KUKA KRL program: Machining.src

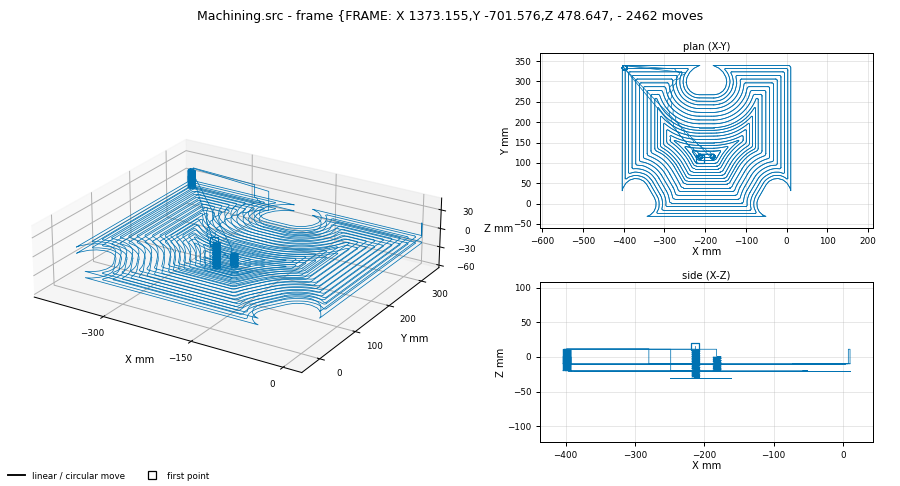
[picture p0: tool path of Machining.src in frame {FRAME: X 1373.155,Y -701.576,Z 478.647,, 2462 of 2464 moves have a stored position in this frame; points joined in program order, loops and branches not executed]
&ACCESS RVP
&REL 1
&PARAM TEMPLATE = C:\KRC\Roboter\Template\vorgabe
&PARAM EDITMASK = *
DEF Machining ( )

; External program calls:
EXT Machining1()


EXT BAS (BAS_COMMAND :IN,REAL :IN )

;FOLD INI
BAS (#INITMOV,0 )
;ENDFOLD (INI)

;FOLD STARTPOS
$BWDSTART = FALSE
PDAT_ACT = PDEFAULT
BAS(#PTP_DAT)
FDAT_ACT = {TOOL_NO 0,BASE_NO 0,IPO_FRAME #BASE}
BAS(#FRAMES)
;ENDFOLD

;FOLD SET DEFAULT SPEED
$VEL.CP=0.2
BAS(#VEL_PTP,100)
BAS(#TOOL,0)
BAS(#BASE,0)
;ENDFOLD

$ADVANCE = 5

PTP $AXIS_ACT ; skip BCO quickly

; Program generated by RoboDK v3.5.4 for GIGASHEEN on 08/07/2019 07:57:20
; Using nominal kinematics.
$APO.CPTP = 1.000
$APO.CDIS = 1.000
$BASE = {FRAME: X 1373.155,Y -701.576,Z 478.647,A -180.000,B 0.620,C 1.380}
$TOOL = {FRAME: X 337.715,Y -2.199,Z 160.575,A 0.000,B 90.000,C 0.000}
; Show 1/2" End Mill TCP
Wait for StrClear($LOOP_MSG[])
$LOOP_CONT = TRUE
$LOOP_MSG[] = "/'1001'"
Wait for StrClear($LOOP_MSG[])
$LOOP_CONT = TRUE
$LOOP_MSG[] = "/''"
Wait for StrClear($LOOP_MSG[])
$LOOP_CONT = TRUE
$LOOP_MSG[] = "/'Pocket2'"
$VEL.CP = 1.00000
$VEL.CP = 1.00000
PTP {A1 32.59641,A2 -47.79719,A3 105.13818,A4 -142.99270,A5 63.54911,A6 162.42451} C_PTP
LIN {X -212.831,Y 109.367,Z 15.000,A 0.015,B 0.000,C 180.000} C_DIS
LIN {X -212.831,Y 109.367,Z 15.000,A 0.015,B 0.000,C 180.000} C_DIS
$VEL.CP = 1.00000
LIN {X -212.831,Y 109.367,Z 11.769,A 0.015,B 0.000,C 180.000} C_DIS
$VEL.CP = 0.10000
LIN {X -212.669,Y 109.348,Z 11.147,A 0.015,B 0.000,C -180.000} C_DIS
LIN {X -212.223,Y 109.320,Z 10.684,A 0.015,B 0.000,C -180.000} C_DIS
LIN {X -211.608,Y 109.335,Z 10.500,A 0.015,B -0.000,C 180.000} C_DIS
LIN {X -206.370,Y 113.359,Z 10.256,A 0.015,B 0.000,C -180.000} C_DIS
LIN {X -207.958,Y 119.769,Z 10.012,A 0.015,B 0.000,C -180.000} C_DIS
LIN {X -214.467,Y 120.884,Z 9.768,A 0.015,B 0.000,C -180.000} C_DIS
LIN {X -218.097,Y 115.366,Z 9.524,A 0.015,B 0.000,C -180.000} C_DIS
LIN {X -214.496,Y 109.830,Z 9.280,A 0.015,B 0.000,C 180.000} C_DIS
LIN {X -207.981,Y 110.910,Z 9.036,A 0.015,B 0.000,C 180.000} C_DIS
LIN {X -206.360,Y 117.312,Z 8.792,A 0.015,B -0.000,C 180.000} C_DIS
LIN {X -211.576,Y 121.363,Z 8.548,A 0.015,B 0.000,C 180.000} C_DIS
LIN {X -217.378,Y 118.207,Z 8.304,A 0.015,B 0.000,C -180.000} C_DIS
LIN {X -216.811,Y 111.627,Z 8.060,A 0.015,B 0.000,C 180.000} C_DIS
LIN {X -210.555,Y 109.510,Z 7.815,A 0.015,B 0.000,C 180.000} C_DIS
LIN {X -206.108,Y 114.393,Z 7.571,A 0.015,B 0.000,C -180.000} C_DIS
LIN {X -208.800,Y 120.423,Z 7.327,A 0.015,B 0.000,C 180.000} C_DIS
LIN {X -215.404,Y 120.374,Z 7.083,A 0.015,B 0.000,C 180.000} C_DIS
LIN {X -218.005,Y 114.303,Z 6.839,A 0.015,B 0.000,C 180.000} C_DIS
LIN {X -213.486,Y 109.488,Z 6.595,A 0.015,B 0.000,C -180.000} C_DIS
LIN {X -207.263,Y 111.699,Z 6.351,A 0.015,B 0.000,C 180.000} C_DIS
LIN {X -206.795,Y 118.286,Z 6.107,A 0.015,B 0.000,C 180.000} C_DIS
LIN {X -212.643,Y 121.355,Z 5.863,A 0.015,B 0.000,C -180.000} C_DIS
LIN {X -217.798,Y 117.227,Z 5.619,A 0.015,B 0.000,C 180.000} C_DIS
LIN {X -216.081,Y 110.849,Z 5.375,A 0.015,B 0.000,C -180.000} C_DIS
LIN {X -209.550,Y 109.867,Z 5.131,A 0.015,B 0.000,C -180.000} C_DIS
LIN {X -206.033,Y 115.457,Z 4.887,A 0.015,B 0.000,C 180.000} C_DIS
LIN {X -209.745,Y 120.919,Z 4.643,A 0.015,B -0.000,C 180.000} C_DIS
LIN {X -216.237,Y 119.707,Z 4.399,A 0.015,B 0.000,C -180.000} C_DIS
LIN {X -217.728,Y 113.273,Z 4.155,A 0.015,B 0.000,C -180.000} C_DIS
LIN {X -212.431,Y 109.329,Z 3.911,A 0.015,B 0.000,C 180.000} C_DIS
LIN {X -206.695,Y 112.602,Z 3.667,A 0.015,B 0.000,C 180.000} C_DIS
LIN {X -207.394,Y 119.169,Z 3.423,A 0.015,B 0.000,C 180.000} C_DIS
LIN {X -213.691,Y 121.159,Z 3.179,A 0.015,B -0.000,C 180.000} C_DIS
LIN {X -218.039,Y 116.188,Z 2.935,A 0.015,B 0.000,C 180.000} C_DIS
LIN {X -215.225,Y 110.212,Z 2.690,A 0.015,B -0.000,C -180.000} C_DIS
LIN {X -208.624,Y 110.395,Z 2.446,A 0.015,B -0.000,C -180.000} C_DIS
LIN {X -206.146,Y 116.517,Z 2.202,A 0.015,B 0.000,C -180.000} C_DIS
LIN {X -210.762,Y 121.241,Z 1.958,A 0.015,B 0.000,C -180.000} C_DIS
LIN {X -216.939,Y 118.904,Z 1.714,A 0.015,B -0.000,C -180.000} C_DIS
LIN {X -217.274,Y 112.308,Z 1.470,A 0.015,B 0.000,C 180.000} C_DIS
LIN {X -211.365,Y 109.359,Z 1.226,A 0.015,B 0.000,C -180.000} C_DIS
LIN {X -206.294,Y 113.590,Z 0.982,A 0.015,B 0.000,C 180.000} C_DIS
LIN {X -208.140,Y 119.932,Z 0.738,A 0.015,B -0.000,C 180.000} C_DIS
LIN {X -214.689,Y 120.782,Z 0.494,A 0.015,B 0.000,C -180.000} C_DIS
LIN {X -218.093,Y 115.122,Z 0.250,A 0.015,B 0.000,C -180.000} C_DIS
LIN {X -214.271,Y 109.736,Z 0.006,A 0.015,B 0.000,C 180.000} C_DIS
LIN {X -207.805,Y 111.079,Z -0.238,A 0.015,B 0.000,C 180.000} C_DIS
LIN {X -206.444,Y 117.541,Z -0.482,A 0.015,B -0.000,C 180.000} C_DIS
LIN {X -211.820,Y 121.378,Z -0.726,A 0.015,B -0.000,C 180.000} C_DIS
LIN {X -217.489,Y 117.990,Z -0.970,A 0.015,B 0.000,C -180.000} C_DIS
LIN {X -216.657,Y 111.438,Z -1.214,A 0.015,B 0.000,C -180.000} C_DIS
LIN {X -210.320,Y 109.575,Z -1.458,A 0.015,B 0.000,C -180.000} C_DIS
LIN {X -206.075,Y 114.634,Z -1.702,A 0.015,B 0.000,C 180.000} C_DIS
LIN {X -209.008,Y 120.551,Z -1.946,A 0.015,B -0.000,C 180.000} C_DIS
LIN {X -215.605,Y 120.235,Z -2.190,A 0.015,B -0.000,C -180.000} C_DIS
LIN {X -217.958,Y 114.064,Z -2.435,A 0.015,B 0.000,C 180.000} C_DIS
LIN {X -213.248,Y 109.435,Z -2.679,A 0.015,B 0.000,C -180.000} C_DIS
LIN {X -207.119,Y 111.896,Z -2.923,A 0.015,B 0.000,C -180.000} C_DIS
LIN {X -206.918,Y 118.497,Z -3.167,A 0.015,B 0.000,C -180.000} C_DIS
LIN {X -212.885,Y 121.327,Z -3.411,A 0.015,B 0.000,C 180.000} C_DIS
LIN {X -217.869,Y 116.993,Z -3.655,A 0.015,B 0.000,C -180.000} C_DIS
LIN {X -215.896,Y 110.691,Z -3.899,A 0.015,B 0.000,C -180.000} C_DIS
LIN {X -209.331,Y 109.973,Z -4.143,A 0.015,B -0.000,C -180.000} C_DIS
LIN {X -206.042,Y 115.700,Z -4.387,A 0.015,B -0.000,C -180.000} C_DIS
LIN {X -209.972,Y 121.008,Z -4.631,A 0.015,B 0.000,C 180.000} C_DIS
LIN {X -216.410,Y 119.535,Z -4.875,A 0.015,B 0.000,C -180.000} C_DIS
LIN {X -217.640,Y 113.046,Z -5.119,A 0.015,B 0.000,C -180.000} C_DIS
LIN {X -212.187,Y 109.319,Z -5.363,A 0.015,B 0.000,C -180.000} C_DIS
LIN {X -206.588,Y 112.821,Z -5.607,A 0.015,B 0.000,C 180.000} C_DIS
LIN {X -207.552,Y 119.354,Z -5.851,A 0.015,B 0.000,C -180.000} C_DIS
LIN {X -213.925,Y 121.089,Z -6.095,A 0.015,B 0.000,C -180.000} C_DIS
LIN {X -218.068,Y 115.945,Z -6.339,A 0.015,B 0.000,C -180.000} C_DIS
LIN {X -215.015,Y 110.089,Z -6.583,A 0.015,B -0.000,C 180.000} C_DIS
LIN {X -208.426,Y 110.539,Z -6.827,A 0.015,B 0.000,C -180.000} C_DIS
LIN {X -206.198,Y 116.756,Z -7.071,A 0.015,B 0.000,C 180.000} C_DIS
LIN {X -211.001,Y 121.288,Z -7.315,A 0.015,B 0.000,C 180.000} C_DIS
LIN {X -217.079,Y 118.704,Z -7.560,A 0.015,B -0.000,C -180.000} C_DIS
LIN {X -217.147,Y 112.100,Z -7.804,A 0.015,B -0.000,C -180.000} C_DIS
LIN {X -211.123,Y 109.392,Z -8.048,A 0.015,B 0.000,C -180.000} C_DIS
LIN {X -206.228,Y 113.825,Z -8.292,A 0.015,B 0.000,C -180.000} C_DIS
LIN {X -208.328,Y 120.087,Z -8.536,A 0.015,B -0.000,C -180.000} C_DIS
LIN {X -214.907,Y 120.671,Z -8.780,A 0.015,B 0.000,C -180.000} C_DIS
LIN {X -218.078,Y 114.879,Z -9.024,A 0.015,B -0.000,C -180.000} C_DIS
LIN {X -214.042,Y 109.651,Z -9.268,A 0.015,B 0.000,C 180.000} C_DIS
LIN {X -207.636,Y 111.255,Z -9.512,A 0.015,B 0.000,C 180.000} C_DIS
LIN {X -206.537,Y 117.767,Z -9.756,A 0.015,B 0.000,C -180.000} C_DIS
LIN {X -212.064,Y 121.383,Z -10.000,A 0.015,B 0.000,C -180.000} C_DIS
LIN {X -213.992,Y 121.383,Z -10.000,A 0.015,B 0.000,C -180.000} C_DIS
CIRC {X -215.914,Y 120.274,Z -10.000,A 0.015,B 0.000,C 180.000},{X -215.915,Y 118.055,Z -10.000,A 0.015,B 0.000,C -180.000} C_DIS
LIN {X -214.810,Y 116.136,Z -10.000,A 0.015,B -0.000,C -180.000} C_DIS
CIRC {X -213.771,Y 115.096,Z -10.000,A 0.015,B 0.000,C 180.000},{X -212.350,Y 114.715,Z -10.000,A 0.015,B 0.000,C 180.000} C_DIS
LIN {X -181.148,Y 114.715,Z -10.000,A 0.015,B 0.000,C 180.000} C_DIS
CIRC {X -179.729,Y 115.095,Z -10.000,A 0.015,B -0.000,C 180.000},{X -178.690,Y 116.133,Z -10.000,A 0.015,B 0.000,C -180.000} C_DIS
LIN {X -177.582,Y 118.050,Z -10.000,A 0.015,B 0.000,C 180.000} C_DIS
CIRC {X -177.581,Y 120.268,Z -10.000,A 0.015,B 0.000,C -180.000},{X -179.502,Y 121.378,Z -10.000,A 0.015,B 0.000,C -180.000} C_DIS
LIN {X -212.064,Y 121.383,Z -10.000,A 0.015,B 0.000,C -180.000} C_DIS
CIRC {X -215.545,Y 122.470,Z -10.000,A 0.015,B 0.000,C 180.000},{X -217.792,Y 125.344,Z -10.000,A 0.015,B -0.000,C -180.000} C_DIS
CIRC {X -219.970,Y 128.243,Z -10.000,A 0.015,B 0.000,C 180.000},{X -223.364,Y 129.521,Z -10.000,A 0.015,B 0.000,C 180.000} C_DIS
CIRC {X -226.438,Y 129.779,Z -10.000,A 0.015,B 0.000,C -180.000},{X -229.509,Y 130.077,Z -10.000,A 0.015,B 0.000,C -180.000} C_DIS
CIRC {X -231.315,Y 129.159,Z -10.000,A 0.015,B 0.000,C -180.000},{X -231.219,Y 127.135,Z -10.000,A 0.015,B 0.000,C 180.000} C_DIS
CIRC {X -228.507,Y 123.213,Z -10.000,A 0.015,B 0.000,C 180.000},{X -225.924,Y 119.206,Z -10.000,A 0.015,B -0.000,C 180.000} C_DIS
CIRC {X -223.440,Y 115.136,Z -10.000,A 0.015,B 0.000,C 180.000},{X -221.024,Y 111.025,Z -10.000,A 0.015,B 0.000,C -180.000} C_DIS
CIRC {X -217.920,Y 107.917,Z -10.000,A 0.015,B -0.000,C 180.000},{X -213.676,Y 106.779,Z -10.000,A 0.015,B 0.000,C 180.000} C_DIS
LIN {X -179.836,Y 106.779,Z -10.000,A 0.015,B 0.000,C 180.000} C_DIS
CIRC {X -175.587,Y 107.917,Z -10.000,A 0.015,B 0.000,C 180.000},{X -172.475,Y 111.026,Z -10.000,A 0.015,B 0.000,C -180.000} C_DIS
CIRC {X -170.064,Y 115.135,Z -10.000,A 0.015,B 0.000,C 180.000},{X -167.600,Y 119.211,Z -10.000,A 0.015,B 0.000,C 180.000} C_DIS
CIRC {X -165.032,Y 123.224,Z -10.000,A 0.015,B 0.000,C 180.000},{X -162.314,Y 127.136,Z -10.000,A 0.015,B 0.000,C 180.000} C_DIS
CIRC {X -162.208,Y 129.160,Z -10.000,A 0.015,B 0.000,C 180.000},{X -164.009,Y 130.087,Z -10.000,A 0.015,B 0.000,C -180.000} C_DIS
CIRC {X -167.842,Y 129.694,Z -10.000,A 0.015,B 0.000,C -180.000},{X -171.671,Y 129.271,Z -10.000,A 0.015,B 0.000,C 180.000} C_DIS
CIRC {X -175.512,Y 128.943,Z -10.000,A 0.015,B -0.000,C -180.000},{X -179.364,Y 128.834,Z -10.000,A 0.015,B 0.000,C 180.000} C_DIS
LIN {X -205.629,Y 128.838,Z -10.000,A 0.015,B 0.000,C -180.000} C_DIS
CIRC {X -214.503,Y 129.009,Z -10.000,A 0.015,B 0.000,C -180.000},{X -223.364,Y 129.521,Z -10.000,A 0.015,B 0.000,C -180.000} C_DIS
CIRC {X -226.590,Y 130.783,Z -10.000,A 0.015,B 0.000,C 180.000},{X -228.564,Y 133.630,Z -10.000,A 0.015,B -0.000,C -180.000} C_DIS
CIRC {X -230.489,Y 136.492,Z -10.000,A 0.015,B 0.000,C -180.000},{X -233.646,Y 137.883,Z -10.000,A 0.015,B 0.000,C -180.000} C_DIS
CIRC {X -239.011,Y 138.684,Z -10.000,A 0.015,B -0.000,C -180.000},{X -244.350,Y 139.648,Z -10.000,A 0.015,B 0.000,C 180.000} C_DIS
CIRC {X -245.188,Y 139.826,Z -10.000,A 0.015,B 0.000,C 180.000},{X -246.019,Y 140.030,Z -10.000,A 0.015,B 0.000,C 180.000} C_DIS
CIRC {X -246.851,Y 140.234,Z -10.000,A 0.015,B 0.000,C -180.000},{X -247.688,Y 140.411,Z -10.000,A 0.015,B -0.000,C 180.000} C_DIS
CIRC {X -249.425,Y 139.627,Z -10.000,A 0.015,B 0.000,C -180.000},{X -249.254,Y 137.730,Z -10.000,A 0.015,B 0.000,C -180.000} C_DIS
CIRC {X -245.418,Y 133.290,Z -10.000,A 0.015,B 0.000,C 180.000},{X -241.535,Y 128.891,Z -10.000,A 0.015,B -0.000,C 180.000} C_DIS
CIRC {X -237.771,Y 124.386,Z -10.000,A 0.015,B 0.000,C -180.000},{X -234.304,Y 119.648,Z -10.000,A 0.015,B -0.000,C 180.000} C_DIS
CIRC {X -231.839,Y 115.776,Z -10.000,A 0.015,B 0.000,C -180.000},{X -229.634,Y 111.750,Z -10.000,A 0.015,B 0.000,C 180.000} C_DIS
CIRC {X -227.507,Y 107.684,Z -10.000,A 0.015,B 0.000,C -180.000},{X -225.271,Y 103.678,Z -10.000,A 0.015,B 0.000,C 180.000} C_DIS
CIRC {X -222.166,Y 100.569,Z -10.000,A 0.015,B 0.000,C 180.000},{X -217.922,Y 99.431,Z -10.000,A 0.015,B -0.000,C 180.000} C_DIS
LIN {X -175.596,Y 99.431,Z -10.000,A 0.015,B 0.000,C -180.000} C_DIS
CIRC {X -171.347,Y 100.569,Z -10.000,A 0.015,B -0.000,C 180.000},{X -168.235,Y 103.679,Z -10.000,A 0.015,B 0.000,C -180.000} C_DIS
CIRC {X -164.238,Y 110.524,Z -10.000,A 0.015,B 0.000,C -180.000},{X -160.181,Y 117.333,Z -10.000,A 0.015,B 0.000,C 180.000} C_DIS
CIRC {X -155.834,Y 123.968,Z -10.000,A 0.015,B 0.000,C 180.000},{X -150.994,Y 130.253,Z -10.000,A 0.015,B 0.000,C -180.000} C_DIS
CIRC {X -149.353,Y 132.160,Z -10.000,A 0.015,B -0.000,C 180.000},{X -147.652,Y 134.012,Z -10.000,A 0.015,B 0.000,C -180.000} C_DIS
CIRC {X -145.937,Y 135.852,Z -10.000,A 0.015,B 0.000,C 180.000},{X -144.257,Y 137.724,Z -10.000,A 0.015,B 0.000,C -180.000} C_DIS
CIRC {X -144.062,Y 139.614,Z -10.000,A 0.015,B 0.000,C 180.000},{X -145.784,Y 140.416,Z -10.000,A 0.015,B 0.000,C 180.000} C_DIS
CIRC {X -154.123,Y 138.916,Z -10.000,A 0.015,B 0.000,C 180.000},{X -162.475,Y 137.498,Z -10.000,A 0.015,B -0.000,C -180.000} C_DIS
CIRC {X -170.891,Y 136.464,Z -10.000,A 0.015,B 0.000,C -180.000},{X -179.363,Y 136.119,Z -10.000,A 0.015,B 0.000,C -180.000} C_DIS
LIN {X -211.942,Y 136.310,Z -10.000,A 0.015,B 0.000,C -180.000} C_DIS
CIRC {X -222.818,Y 136.767,Z -10.000,A 0.015,B 0.000,C -180.000},{X -233.646,Y 137.883,Z -10.000,A 0.015,B 0.000,C -180.000} C_DIS
CIRC {X -236.389,Y 139.137,Z -10.000,A 0.015,B 0.000,C -180.000},{X -237.966,Y 141.708,Z -10.000,A 0.015,B 0.000,C 180.000} C_DIS
CIRC {X -239.496,Y 144.291,Z -10.000,A 0.015,B 0.000,C -180.000},{X -242.167,Y 145.662,Z -10.000,A 0.015,B 0.000,C 180.000} C_DIS
CIRC {X -243.731,Y 145.978,Z -10.000,A 0.015,B 0.000,C -180.000},{X -245.290,Y 146.311,Z -10.000,A 0.015,B 0.000,C 180.000} C_DIS
CIRC {X -260.066,Y 150.251,Z -10.000,A 0.015,B 0.000,C -180.000},{X -274.434,Y 155.484,Z -10.000,A 0.015,B 0.000,C 180.000} C_DIS
CIRC {X -275.992,Y 154.954,Z -10.000,A 0.015,B 0.000,C 180.000},{X -275.665,Y 153.341,Z -10.000,A 0.015,B 0.000,C -180.000} C_DIS
CIRC {X -256.299,Y 136.003,Z -10.000,A 0.015,B 0.000,C -180.000},{X -239.991,Y 115.762,Z -10.000,A 0.015,B -0.000,C -180.000} C_DIS
CIRC {X -237.062,Y 111.161,Z -10.000,A 0.015,B 0.000,C -180.000},{X -234.439,Y 106.379,Z -10.000,A 0.015,B 0.000,C -180.000} C_DIS
CIRC {X -231.910,Y 101.549,Z -10.000,A 0.015,B 0.000,C 180.000},{X -229.251,Y 96.790,Z -10.000,A 0.015,B 0.000,C -180.000} C_DIS
CIRC {X -226.146,Y 93.681,Z -10.000,A 0.015,B 0.000,C -180.000},{X -221.903,Y 92.543,Z -10.000,A 0.015,B 0.000,C 180.000} C_DIS
LIN {X -171.621,Y 92.543,Z -10.000,A 0.015,B 0.000,C 180.000} C_DIS
CIRC {X -167.372,Y 93.681,Z -10.000,A 0.015,B -0.000,C 180.000},{X -164.260,Y 96.791,Z -10.000,A 0.015,B 0.000,C -180.000} C_DIS
LIN {X -155.690,Y 111.783,Z -10.000,A 0.015,B -0.000,C -180.000} C_DIS
CIRC {X -151.103,Y 119.108,Z -10.000,A 0.015,B 0.000,C 180.000},{X -145.877,Y 125.992,Z -10.000,A 0.015,B 0.000,C -180.000} C_DIS
CIRC {X -139.411,Y 133.389,Z -10.000,A 0.015,B 0.000,C -180.000},{X -132.597,Y 140.468,Z -10.000,A 0.015,B 0.000,C -180.000} C_DIS
CIRC {X -125.399,Y 147.158,Z -10.000,A 0.015,B 0.000,C -180.000},{X -117.791,Y 153.378,Z -10.000,A 0.015,B 0.000,C 180.000} C_DIS
CIRC {X -117.471,Y 154.991,Z -10.000,A 0.015,B 0.000,C -180.000},{X -119.032,Y 155.512,Z -10.000,A 0.015,B -0.000,C 180.000} C_DIS
CIRC {X -144.718,Y 147.150,Z -10.000,A 0.015,B 0.000,C 180.000},{X -171.448,Y 143.251,Z -10.000,A 0.015,B 0.000,C -180.000} C_DIS
LIN {X -214.915,Y 143.013,Z -10.000,A 0.015,B 0.000,C -180.000} C_DIS
CIRC {X -228.606,Y 143.678,Z -10.000,A 0.015,B 0.000,C 180.000},{X -242.167,Y 145.662,Z -10.000,A 0.015,B 0.000,C 180.000} C_DIS
CIRC {X -244.832,Y 147.079,Z -10.000,A 0.015,B 0.000,C 180.000},{X -246.259,Y 149.738,Z -10.000,A 0.015,B 0.000,C -180.000} C_DIS
CIRC {X -247.644,Y 152.406,Z -10.000,A 0.015,B 0.000,C 180.000},{X -250.236,Y 153.926,Z -10.000,A 0.015,B 0.000,C 180.000} C_DIS
CIRC {X -267.068,Y 159.341,Z -10.000,A 0.015,B 0.000,C -180.000},{X -283.104,Y 166.788,Z -10.000,A 0.015,B 0.000,C 180.000} C_DIS
CIRC {X -285.347,Y 166.742,Z -10.000,A 0.015,B 0.000,C 180.000},{X -286.456,Y 164.791,Z -10.000,A 0.015,B 0.000,C 180.000} C_DIS
LIN {X -286.456,Y 156.656,Z -10.000,A 0.015,B 0.000,C 180.000} C_DIS
CIRC {X -285.697,Y 153.532,Z -10.000,A 0.015,B -0.000,C 180.000},{X -283.591,Y 151.104,Z -10.000,A 0.015,B 0.000,C 180.000} C_DIS
CIRC {X -262.735,Y 133.303,Z -10.000,A 0.015,B -0.000,C 180.000},{X -245.343,Y 112.104,Z -10.000,A 0.015,B 0.000,C -180.000} C_DIS
CIRC {X -241.977,Y 106.818,Z -10.000,A 0.015,B 0.000,C 180.000},{X -238.961,Y 101.324,Z -10.000,A 0.015,B 0.000,C -180.000} C_DIS
CIRC {X -236.053,Y 95.776,Z -10.000,A 0.015,B 0.000,C -180.000},{X -232.998,Y 90.307,Z -10.000,A 0.015,B 0.000,C 180.000} C_DIS
CIRC {X -229.893,Y 87.199,Z -10.000,A 0.015,B -0.000,C 180.000},{X -225.649,Y 86.061,Z -10.000,A 0.015,B 0.000,C -180.000} C_DIS
LIN {X -167.880,Y 86.061,Z -10.000,A 0.015,B 0.000,C -180.000} C_DIS
CIRC {X -163.631,Y 87.199,Z -10.000,A 0.015,B 0.000,C 180.000},{X -160.519,Y 90.308,Z -10.000,A 0.015,B -0.000,C -180.000} C_DIS
CIRC {X -155.909,Y 98.378,Z -10.000,A 0.015,B 0.000,C -180.000},{X -151.379,Y 106.494,Z -10.000,A 0.015,B 0.000,C -180.000} C_DIS
CIRC {X -146.502,Y 114.418,Z -10.000,A 0.015,B 0.000,C -180.000},{X -140.895,Y 121.844,Z -10.000,A 0.015,B -0.000,C -180.000} C_DIS
CIRC {X -133.849,Y 129.861,Z -10.000,A 0.015,B 0.000,C 180.000},{X -126.384,Y 137.490,Z -10.000,A 0.015,B 0.000,C 180.000} C_DIS
CIRC {X -118.431,Y 144.615,Z -10.000,A 0.015,B 0.000,C -180.000},{X -109.947,Y 151.097,Z -10.000,A 0.015,B 0.000,C -180.000} C_DIS
CIRC {X -107.822,Y 153.530,Z -10.000,A 0.015,B -0.000,C 180.000},{X -107.056,Y 156.667,Z -10.000,A 0.015,B 0.000,C -180.000} C_DIS
LIN {X -107.057,Y 164.754,Z -10.000,A 0.015,B -0.000,C 180.000} C_DIS
CIRC {X -108.165,Y 166.709,Z -10.000,A 0.015,B 0.000,C -180.000},{X -110.412,Y 166.762,Z -10.000,A 0.015,B 0.000,C -180.000} C_DIS
CIRC {X -124.973,Y 159.992,Z -10.000,A 0.015,B 0.000,C -180.000},{X -140.210,Y 154.923,Z -10.000,A 0.015,B 0.000,C -180.000} C_DIS
CIRC {X -155.898,Y 151.522,Z -10.000,A 0.015,B -0.000,C 180.000},{X -171.849,Y 149.721,Z -10.000,A 0.015,B 0.000,C 180.000} C_DIS
LIN {X -214.914,Y 149.495,Z -10.000,A 0.015,B 0.000,C 180.000} C_DIS
CIRC {X -232.714,Y 150.608,Z -10.000,A 0.015,B 0.000,C -180.000},{X -250.236,Y 153.926,Z -10.000,A 0.015,B -0.000,C -180.000} C_DIS
CIRC {X -253.513,Y 155.921,Z -10.000,A 0.015,B 0.000,C 180.000},{X -255.110,Y 159.408,Z -10.000,A 0.015,B 0.000,C -180.000} C_DIS
CIRC {X -256.625,Y 162.907,Z -10.000,A 0.015,B 0.000,C -180.000},{X -259.752,Y 165.088,Z -10.000,A 0.015,B 0.000,C 180.000} C_DIS
CIRC {X -271.740,Y 169.872,Z -10.000,A 0.015,B -0.000,C -180.000},{X -283.226,Y 175.760,Z -10.000,A 0.015,B 0.000,C 180.000} C_DIS
CIRC {X -285.285,Y 177.012,Z -10.000,A 0.015,B 0.000,C 180.000},{X -287.272,Y 178.375,Z -10.000,A 0.015,B 0.000,C 180.000} C_DIS
CIRC {X -289.236,Y 179.770,Z -10.000,A 0.015,B 0.000,C -180.000},{X -291.232,Y 181.119,Z -10.000,A 0.015,B 0.000,C 180.000} C_DIS
CIRC {X -293.404,Y 181.215,Z -10.000,A 0.015,B 0.000,C -180.000},{X -294.518,Y 179.349,Z -10.000,A 0.015,B 0.000,C 180.000} C_DIS
LIN {X -294.517,Y 153.793,Z -10.000,A 0.015,B 0.000,C 180.000} C_DIS
CIRC {X -293.420,Y 149.385,Z -10.000,A 0.015,B 0.000,C 180.000},{X -290.385,Y 146.007,Z -10.000,A 0.015,B 0.000,C -180.000} C_DIS
CIRC {X -279.458,Y 137.810,Z -10.000,A 0.015,B 0.000,C 180.000},{X -269.378,Y 128.592,Z -10.000,A 0.015,B 0.000,C -180.000} C_DIS
CIRC {X -260.210,Y 118.469,Z -10.000,A 0.015,B 0.000,C 180.000},{X -251.999,Y 107.556,Z -10.000,A 0.015,B 0.000,C 180.000} C_DIS
LIN {X -237.657,Y 82.245,Z -10.000,A 0.015,B 0.000,C 180.000} C_DIS
CIRC {X -234.552,Y 79.137,Z -10.000,A 0.015,B 0.000,C -180.000},{X -230.308,Y 77.999,Z -10.000,A 0.015,B 0.000,C 180.000} C_DIS
LIN {X -163.228,Y 77.999,Z -10.000,A 0.015,B 0.000,C 180.000} C_DIS
CIRC {X -158.979,Y 79.137,Z -10.000,A 0.015,B -0.000,C -180.000},{X -155.867,Y 82.246,Z -10.000,A 0.015,B 0.000,C -180.000} C_DIS
LIN {X -143.614,Y 103.306,Z -10.000,A 0.015,B 0.000,C 180.000} C_DIS
CIRC {X -136.952,Y 113.522,Z -10.000,A 0.015,B 0.000,C -180.000},{X -129.342,Y 123.053,Z -10.000,A 0.015,B -0.000,C -180.000} C_DIS
CIRC {X -116.981,Y 135.379,Z -10.000,A 0.015,B -0.000,C -180.000},{X -103.127,Y 146.001,Z -10.000,A 0.015,B 0.000,C 180.000} C_DIS
CIRC {X -100.092,Y 149.354,Z -10.000,A 0.015,B -0.000,C 180.000},{X -98.994,Y 153.742,Z -10.000,A 0.015,B 0.000,C -180.000} C_DIS
LIN {X -98.995,Y 179.303,Z -10.000,A 0.015,B 0.000,C 180.000} C_DIS
CIRC {X -100.110,Y 181.183,Z -10.000,A 0.015,B 0.000,C 180.000},{X -102.295,Y 181.107,Z -10.000,A 0.015,B 0.000,C 180.000} C_DIS
LIN {X -112.706,Y 174.512,Z -10.000,A 0.015,B 0.000,C -180.000} C_DIS
CIRC {X -118.053,Y 171.438,Z -10.000,A 0.015,B 0.000,C -180.000},{X -123.617,Y 168.779,Z -10.000,A 0.015,B 0.000,C -180.000} C_DIS
CIRC {X -135.372,Y 164.377,Z -10.000,A 0.015,B 0.000,C -180.000},{X -147.504,Y 161.160,Z -10.000,A 0.015,B 0.000,C 180.000} C_DIS
CIRC {X -159.863,Y 159.005,Z -10.000,A 0.015,B 0.000,C 180.000},{X -172.347,Y 157.768,Z -10.000,A 0.015,B -0.000,C -180.000} C_DIS
LIN {X -214.913,Y 157.557,Z -10.000,A 0.015,B 0.000,C 180.000} C_DIS
CIRC {X -237.646,Y 159.455,Z -10.000,A 0.015,B 0.000,C 180.000},{X -259.752,Y 165.088,Z -10.000,A 0.015,B -0.000,C 180.000} C_DIS
CIRC {X -262.782,Y 167.298,Z -10.000,A 0.015,B 0.000,C -180.000},{X -264.055,Y 170.825,Z -10.000,A 0.015,B 0.000,C 180.000} C_DIS
CIRC {X -265.246,Y 174.357,Z -10.000,A 0.015,B 0.000,C 180.000},{X -268.112,Y 176.739,Z -10.000,A 0.015,B 0.000,C 180.000} C_DIS
CIRC {X -273.836,Y 179.444,Z -10.000,A 0.015,B 0.000,C 180.000},{X -279.423,Y 182.421,Z -10.000,A 0.015,B 0.000,C 180.000} C_DIS
CIRC {X -284.615,Y 185.584,Z -10.000,A 0.015,B 0.000,C -180.000},{X -289.619,Y 189.036,Z -10.000,A 0.015,B 0.000,C -180.000} C_DIS
CIRC {X -294.482,Y 192.681,Z -10.000,A 0.015,B 0.000,C 180.000},{X -299.265,Y 196.430,Z -10.000,A 0.015,B 0.000,C -180.000} C_DIS
CIRC {X -301.327,Y 196.666,Z -10.000,A 0.015,B -0.000,C -180.000},{X -302.432,Y 194.910,Z -10.000,A 0.015,B -0.000,C 180.000} C_DIS
LIN {X -302.430,Y 149.108,Z -10.000,A 0.015,B 0.000,C -180.000} C_DIS
CIRC {X -301.333,Y 144.881,Z -10.000,A 0.015,B -0.000,C -180.000},{X -298.320,Y 141.721,Z -10.000,A 0.015,B 0.000,C 180.000} C_DIS
CIRC {X -286.884,Y 133.713,Z -10.000,A 0.015,B 0.000,C 180.000},{X -276.409,Y 124.483,Z -10.000,A 0.015,B 0.000,C 180.000} C_DIS
CIRC {X -266.954,Y 114.219,Z -10.000,A 0.015,B 0.000,C -180.000},{X -258.532,Y 103.091,Z -10.000,A 0.015,B 0.000,C 180.000} C_DIS
LIN {X -242.230,Y 74.332,Z -10.000,A 0.015,B 0.000,C 180.000} C_DIS
CIRC {X -239.125,Y 71.224,Z -10.000,A 0.015,B 0.000,C -180.000},{X -234.881,Y 70.085,Z -10.000,A 0.015,B 0.000,C -180.000} C_DIS
LIN {X -158.662,Y 70.085,Z -10.000,A 0.015,B -0.000,C -180.000} C_DIS
CIRC {X -154.412,Y 71.224,Z -10.000,A 0.015,B -0.000,C -180.000},{X -151.301,Y 74.333,Z -10.000,A 0.015,B 0.000,C 180.000} C_DIS
LIN {X -138.428,Y 96.769,Z -10.000,A 0.015,B 0.000,C 180.000} C_DIS
CIRC {X -131.453,Y 107.680,Z -10.000,A 0.015,B 0.000,C 180.000},{X -123.402,Y 117.824,Z -10.000,A 0.015,B 0.000,C -180.000} C_DIS
CIRC {X -110.186,Y 130.785,Z -10.000,A 0.015,B 0.000,C -180.000},{X -95.219,Y 141.676,Z -10.000,A 0.015,B -0.000,C 180.000} C_DIS
CIRC {X -92.185,Y 144.865,Z -10.000,A 0.015,B 0.000,C -180.000},{X -91.081,Y 149.126,Z -10.000,A 0.015,B -0.000,C -180.000} C_DIS
LIN {X -91.082,Y 194.877,Z -10.000,A 0.015,B 0.000,C -180.000} C_DIS
CIRC {X -92.187,Y 196.636,Z -10.000,A 0.015,B 0.000,C -180.000},{X -94.252,Y 196.407,Z -10.000,A 0.015,B 0.000,C -180.000} C_DIS
CIRC {X -105.378,Y 188.269,Z -10.000,A 0.015,B 0.000,C 180.000},{X -117.113,Y 181.037,Z -10.000,A 0.015,B 0.000,C 180.000} C_DIS
CIRC {X -129.540,Y 175.034,Z -10.000,A 0.015,B -0.000,C -180.000},{X -142.619,Y 170.630,Z -10.000,A 0.015,B 0.000,C 180.000} C_DIS
CIRC {X -160.452,Y 167.023,Z -10.000,A 0.015,B 0.000,C -180.000},{X -178.596,Y 165.675,Z -10.000,A 0.015,B -0.000,C -180.000} C_DIS
LIN {X -214.912,Y 165.470,Z -10.000,A 0.015,B 0.000,C 180.000} C_DIS
CIRC {X -242.102,Y 168.320,Z -10.000,A 0.015,B 0.000,C -180.000},{X -268.112,Y 176.739,Z -10.000,A 0.015,B 0.000,C 180.000} C_DIS
CIRC {X -270.852,Y 179.121,Z -10.000,A 0.015,B 0.000,C 180.000},{X -271.780,Y 182.630,Z -10.000,A 0.015,B 0.000,C 180.000} C_DIS
CIRC {X -272.624,Y 186.136,Z -10.000,A 0.015,B 0.000,C 180.000},{X -275.178,Y 188.682,Z -10.000,A 0.015,B -0.000,C -180.000} C_DIS
CIRC {X -292.140,Y 200.054,Z -10.000,A 0.015,B -0.000,C 180.000},{X -307.005,Y 214.058,Z -10.000,A 0.015,B 0.000,C 180.000} C_DIS
CIRC {X -308.889,Y 214.518,Z -10.000,A 0.015,B 0.000,C -180.000},{X -309.989,Y 212.920,Z -10.000,A 0.015,B 0.000,C -180.000} C_DIS
LIN {X -309.988,Y 144.412,Z -10.000,A 0.015,B 0.000,C -180.000} C_DIS
CIRC {X -308.891,Y 140.364,Z -10.000,A 0.015,B 0.000,C 180.000},{X -305.900,Y 137.424,Z -10.000,A 0.015,B 0.000,C -180.000} C_DIS
CIRC {X -293.968,Y 129.683,Z -10.000,A 0.015,B -0.000,C -180.000},{X -283.111,Y 120.496,Z -10.000,A 0.015,B 0.000,C -180.000} C_DIS
CIRC {X -273.384,Y 110.134,Z -10.000,A 0.015,B 0.000,C 180.000},{X -264.772,Y 98.827,Z -10.000,A 0.015,B 0.000,C 180.000} C_DIS
LIN {X -246.597,Y 66.775,Z -10.000,A 0.015,B 0.000,C -180.000} C_DIS
CIRC {X -243.492,Y 63.666,Z -10.000,A 0.015,B 0.000,C -180.000},{X -239.248,Y 62.528,Z -10.000,A 0.015,B 0.000,C -180.000} C_DIS
LIN {X -154.301,Y 62.528,Z -10.000,A 0.015,B 0.000,C 180.000} C_DIS
CIRC {X -150.051,Y 63.666,Z -10.000,A 0.015,B 0.000,C -180.000},{X -146.940,Y 66.776,Z -10.000,A 0.015,B 0.000,C -180.000} C_DIS
LIN {X -133.475,Y 90.526,Z -10.000,A 0.015,B 0.000,C 180.000} C_DIS
CIRC {X -126.201,Y 102.100,Z -10.000,A 0.015,B 0.000,C 180.000},{X -117.730,Y 112.830,Z -10.000,A 0.015,B 0.000,C 180.000} C_DIS
CIRC {X -103.683,Y 126.365,Z -10.000,A 0.015,B 0.000,C 180.000},{X -87.612,Y 137.422,Z -10.000,A 0.015,B 0.000,C 180.000} C_DIS
CIRC {X -84.620,Y 140.388,Z -10.000,A 0.015,B 0.000,C 180.000},{X -83.524,Y 144.456,Z -10.000,A 0.015,B -0.000,C 180.000} C_DIS
LIN {X -83.526,Y 212.917,Z -10.000,A 0.015,B 0.000,C 180.000} C_DIS
CIRC {X -84.626,Y 214.525,Z -10.000,A 0.015,B 0.000,C 180.000},{X -86.524,Y 214.081,Z -10.000,A 0.015,B 0.000,C 180.000} C_DIS
CIRC {X -96.057,Y 204.656,Z -10.000,A 0.015,B 0.000,C 180.000},{X -106.492,Y 196.240,Z -10.000,A 0.015,B 0.000,C 180.000} C_DIS
CIRC {X -117.758,Y 188.969,Z -10.000,A 0.015,B 0.000,C -180.000},{X -129.755,Y 182.980,Z -10.000,A 0.015,B 0.000,C -180.000} C_DIS
CIRC {X -150.345,Y 176.312,Z -10.000,A 0.015,B -0.000,C 180.000},{X -171.823,Y 173.644,Z -10.000,A 0.015,B 0.000,C 180.000} C_DIS
LIN {X -214.911,Y 173.027,Z -10.000,A 0.015,B 0.000,C 180.000} C_DIS
CIRC {X -246.044,Y 177.007,Z -10.000,A 0.015,B -0.000,C 180.000},{X -275.178,Y 188.682,Z -10.000,A 0.015,B -0.000,C 180.000} C_DIS
CIRC {X -277.566,Y 191.162,Z -10.000,A 0.015,B 0.000,C 180.000},{X -278.165,Y 194.553,Z -10.000,A 0.015,B 0.000,C -180.000} C_DIS
CIRC {X -278.697,Y 197.935,Z -10.000,A 0.015,B 0.000,C -180.000},{X -280.932,Y 200.530,Z -10.000,A 0.015,B 0.000,C -180.000} C_DIS
CIRC {X -286.576,Y 204.460,Z -10.000,A 0.015,B 0.000,C -180.000},{X -292.005,Y 208.681,Z -10.000,A 0.015,B 0.000,C 180.000} C_DIS
CIRC {X -298.388,Y 214.578,Z -10.000,A 0.015,B -0.000,C 180.000},{X -304.037,Y 221.179,Z -10.000,A 0.015,B 0.000,C -180.000} C_DIS
CIRC {X -309.204,Y 228.148,Z -10.000,A 0.015,B 0.000,C 180.000},{X -314.212,Y 235.232,Z -10.000,A 0.015,B 0.000,C -180.000} C_DIS
CIRC {X -315.961,Y 235.836,Z -10.000,A 0.015,B 0.000,C -180.000},{X -317.059,Y 234.345,Z -10.000,A 0.015,B 0.000,C 180.000} C_DIS
LIN {X -317.056,Y 140.026,Z -10.000,A 0.015,B 0.000,C 180.000} C_DIS
CIRC {X -315.919,Y 135.980,Z -10.000,A 0.015,B 0.000,C 180.000},{X -312.840,Y 133.120,Z -10.000,A 0.015,B 0.000,C 180.000} C_DIS
CIRC {X -300.788,Y 125.887,Z -10.000,A 0.015,B 0.000,C -180.000},{X -289.792,Y 117.133,Z -10.000,A 0.015,B 0.000,C -180.000} C_DIS
CIRC {X -279.970,Y 107.089,Z -10.000,A 0.015,B 0.000,C -180.000},{X -271.382,Y 95.971,Z -10.000,A 0.015,B 0.000,C 180.000} C_DIS
LIN {X -250.665,Y 59.677,Z -10.000,A 0.015,B 0.000,C 180.000} C_DIS
CIRC {X -247.582,Y 56.590,Z -10.000,A 0.015,B 0.000,C 180.000},{X -243.367,Y 55.460,Z -10.000,A 0.015,B 0.000,C -180.000} C_DIS
LIN {X -150.139,Y 55.460,Z -10.000,A 0.015,B 0.000,C -180.000} C_DIS
CIRC {X -145.961,Y 56.578,Z -10.000,A 0.015,B 0.000,C 180.000},{X -142.902,Y 59.636,Z -10.000,A 0.015,B 0.000,C 180.000} C_DIS
LIN {X -124.324,Y 91.782,Z -10.000,A 0.015,B -0.000,C -180.000} C_DIS
CIRC {X -113.008,Y 107.840,Z -10.000,A 0.015,B 0.000,C 180.000},{X -99.006,Y 121.616,Z -10.000,A 0.015,B 0.000,C -180.000} C_DIS
CIRC {X -94.687,Y 124.907,Z -10.000,A 0.015,B 0.000,C 180.000},{X -90.139,Y 127.873,Z -10.000,A 0.015,B -0.000,C 180.000} C_DIS
CIRC {X -85.441,Y 130.592,Z -10.000,A 0.015,B 0.000,C -180.000},{X -80.655,Y 133.151,Z -10.000,A 0.015,B 0.000,C 180.000} C_DIS
CIRC {X -77.588,Y 135.998,Z -10.000,A 0.015,B 0.000,C -180.000},{X -76.455,Y 140.027,Z -10.000,A 0.015,B 0.000,C 180.000} C_DIS
LIN {X -76.458,Y 234.319,Z -10.000,A 0.015,B 0.000,C -180.000} C_DIS
CIRC {X -77.555,Y 235.807,Z -10.000,A 0.015,B 0.000,C 180.000},{X -79.300,Y 235.198,Z -10.000,A 0.015,B 0.000,C -180.000} C_DIS
LIN {X -85.769,Y 225.738,Z -10.000,A 0.015,B -0.000,C -180.000} C_DIS
CIRC {X -89.208,Y 221.090,Z -10.000,A 0.015,B -0.000,C 180.000},{X -92.984,Y 216.711,Z -10.000,A 0.015,B -0.000,C 180.000} C_DIS
CIRC {X -110.064,Y 201.792,Z -10.000,A 0.015,B -0.000,C -180.000},{X -129.856,Y 190.720,Z -10.000,A 0.015,B 0.000,C -180.000} C_DIS
CIRC {X -151.347,Y 183.599,Z -10.000,A 0.015,B 0.000,C -180.000},{X -173.740,Y 180.264,Z -10.000,A 0.015,B 0.000,C 180.000} C_DIS
LIN {X -214.910,Y 180.096,Z -10.000,A 0.015,B 0.000,C 180.000} C_DIS
CIRC {X -235.772,Y 182.015,Z -10.000,A 0.015,B 0.000,C 180.000},{X -255.937,Y 187.701,Z -10.000,A 0.015,B 0.000,C -180.000} C_DIS
CIRC {X -268.781,Y 193.441,Z -10.000,A 0.015,B 0.000,C 180.000},{X -280.932,Y 200.530,Z -10.000,A 0.015,B 0.000,C 180.000} C_DIS
CIRC {X -282.974,Y 202.998,Z -10.000,A 0.015,B 0.000,C 180.000},{X -283.279,Y 206.188,Z -10.000,A 0.015,B 0.000,C 180.000} C_DIS
CIRC {X -283.517,Y 209.363,Z -10.000,A 0.015,B 0.000,C -180.000},{X -285.395,Y 211.936,Z -10.000,A 0.015,B 0.000,C 180.000} C_DIS
CIRC {X -286.589,Y 212.880,Z -10.000,A 0.015,B 0.000,C -180.000},{X -287.772,Y 213.839,Z -10.000,A 0.015,B -0.000,C 180.000} C_DIS
CIRC {X -297.447,Y 222.996,Z -10.000,A 0.015,B 0.000,C 180.000},{X -305.736,Y 233.423,Z -10.000,A 0.015,B 0.000,C -180.000} C_DIS
CIRC {X -312.645,Y 244.798,Z -10.000,A 0.015,B 0.000,C 180.000},{X -318.257,Y 256.865,Z -10.000,A 0.015,B 0.000,C -180.000} C_DIS
CIRC {X -321.429,Y 258.600,Z -10.000,A 0.015,B 0.000,C -180.000},{X -323.731,Y 255.812,Z -10.000,A 0.015,B 0.000,C -180.000} C_DIS
LIN {X -323.728,Y 135.948,Z -10.000,A 0.015,B 0.000,C -180.000} C_DIS
CIRC {X -322.592,Y 131.906,Z -10.000,A 0.015,B -0.000,C -180.000},{X -319.516,Y 129.049,Z -10.000,A 0.015,B 0.000,C 180.000} C_DIS
CIRC {X -315.449,Y 126.976,Z -10.000,A 0.015,B -0.000,C 180.000},{X -311.368,Y 124.929,Z -10.000,A 0.015,B 0.000,C -180.000} C_DIS
CIRC {X -307.363,Y 122.731,Z -10.000,A 0.015,B 0.000,C 180.000},{X -303.548,Y 120.218,Z -10.000,A 0.015,B 0.000,C 180.000} C_DIS
CIRC {X -295.701,Y 113.927,Z -10.000,A 0.015,B 0.000,C -180.000},{X -288.560,Y 106.843,Z -10.000,A 0.015,B -0.000,C -180.000} C_DIS
CIRC {X -282.068,Y 99.172,Z -10.000,A 0.015,B 0.000,C -180.000},{X -276.116,Y 91.074,Z -10.000,A 0.015,B 0.000,C -180.000} C_DIS
LIN {X -254.447,Y 52.849,Z -10.000,A 0.015,B 0.000,C -180.000} C_DIS
CIRC {X -251.558,Y 49.879,Z -10.000,A 0.015,B 0.000,C 180.000},{X -247.561,Y 48.787,Z -10.000,A 0.015,B 0.000,C 180.000} C_DIS
LIN {X -145.882,Y 48.787,Z -10.000,A 0.015,B 0.000,C -180.000} C_DIS
CIRC {X -141.921,Y 49.879,Z -10.000,A 0.015,B 0.000,C -180.000},{X -139.079,Y 52.846,Z -10.000,A 0.015,B 0.000,C 180.000} C_DIS
CIRC {X -129.496,Y 70.166,Z -10.000,A 0.015,B 0.000,C -180.000},{X -119.552,Y 87.282,Z -10.000,A 0.015,B 0.000,C 180.000} C_DIS
CIRC {X -107.953,Y 103.413,Z -10.000,A 0.015,B 0.000,C 180.000},{X -93.747,Y 117.301,Z -10.000,A 0.015,B 0.000,C -180.000} C_DIS
CIRC {X -89.122,Y 120.738,Z -10.000,A 0.015,B -0.000,C 180.000},{X -84.188,Y 123.713,Z -10.000,A 0.015,B 0.000,C 180.000} C_DIS
CIRC {X -79.107,Y 126.414,Z -10.000,A 0.015,B 0.000,C -180.000},{X -73.995,Y 129.059,Z -10.000,A 0.015,B 0.000,C -180.000} C_DIS
CIRC {X -70.920,Y 131.906,Z -10.000,A 0.015,B -0.000,C 180.000},{X -69.783,Y 135.940,Z -10.000,A 0.015,B 0.000,C -180.000} C_DIS
LIN {X -69.786,Y 255.798,Z -10.000,A 0.015,B 0.000,C -180.000} C_DIS
CIRC {X -72.088,Y 258.586,Z -10.000,A 0.015,B 0.000,C -180.000},{X -75.260,Y 256.852,Z -10.000,A 0.015,B 0.000,C 180.000} C_DIS
CIRC {X -85.390,Y 237.376,Z -10.000,A 0.015,B 0.000,C 180.000},{X -99.163,Y 220.282,Z -10.000,A 0.015,B 0.000,C -180.000} C_DIS
CIRC {X -115.992,Y 206.196,Z -10.000,A 0.015,B 0.000,C 180.000},{X -135.206,Y 195.593,Z -10.000,A 0.015,B 0.000,C 180.000} C_DIS
CIRC {X -154.489,Y 189.413,Z -10.000,A 0.015,B 0.000,C 180.000},{X -174.605,Y 187.101,Z -10.000,A 0.015,B -0.000,C 180.000} C_DIS
LIN {X -214.909,Y 186.768,Z -10.000,A 0.015,B 0.000,C -180.000} C_DIS
CIRC {X -234.631,Y 188.589,Z -10.000,A 0.015,B -0.000,C -180.000},{X -253.689,Y 193.983,Z -10.000,A 0.015,B 0.000,C -180.000} C_DIS
CIRC {X -270.205,Y 201.788,Z -10.000,A 0.015,B 0.000,C 180.000},{X -285.395,Y 211.936,Z -10.000,A 0.015,B 0.000,C -180.000} C_DIS
CIRC {X -288.001,Y 215.682,Z -10.000,A 0.015,B -0.000,C -180.000},{X -288.034,Y 220.245,Z -10.000,A 0.015,B 0.000,C -180.000} C_DIS
CIRC {X -287.896,Y 224.757,Z -10.000,A 0.015,B 0.000,C -180.000},{X -290.037,Y 228.730,Z -10.000,A 0.015,B 0.000,C 180.000} C_DIS
CIRC {X -295.052,Y 234.525,Z -10.000,A 0.015,B -0.000,C 180.000},{X -299.547,Y 240.731,Z -10.000,A 0.015,B 0.000,C 180.000} C_DIS
CIRC {X -306.108,Y 252.254,Z -10.000,A 0.015,B 0.000,C -180.000},{X -311.095,Y 264.539,Z -10.000,A 0.015,B -0.000,C -180.000} C_DIS
CIRC {X -313.202,Y 267.414,Z -10.000,A 0.015,B 0.000,C 180.000},{X -316.593,Y 268.510,Z -10.000,A 0.015,B -0.000,C 180.000} C_DIS
LIN {X -329.241,Y 268.510,Z -10.000,A 0.015,B 0.000,C 180.000} C_DIS
CIRC {X -331.966,Y 267.381,Z -10.000,A 0.015,B -0.000,C -180.000},{X -333.094,Y 264.657,Z -10.000,A 0.015,B 0.000,C 180.000} C_DIS
LIN {X -333.091,Y 129.745,Z -10.000,A 0.015,B 0.000,C -180.000} C_DIS
CIRC {X -331.999,Y 125.980,Z -10.000,A 0.015,B -0.000,C 180.000},{X -329.061,Y 123.382,Z -10.000,A 0.015,B -0.000,C -180.000} C_DIS
CIRC {X -321.208,Y 119.456,Z -10.000,A 0.015,B -0.000,C -180.000},{X -313.534,Y 115.191,Z -10.000,A 0.015,B 0.000,C -180.000} C_DIS
CIRC {X -306.224,Y 110.302,Z -10.000,A 0.015,B 0.000,C 180.000},{X -299.557,Y 104.568,Z -10.000,A 0.015,B -0.000,C 180.000} C_DIS
CIRC {X -288.536,Y 92.187,Z -10.000,A 0.015,B 0.000,C -180.000},{X -279.425,Y 78.341,Z -10.000,A 0.015,B 0.000,C -180.000} C_DIS
LIN {X -263.111,Y 49.584,Z -10.000,A 0.015,B 0.000,C 180.000} C_DIS
CIRC {X -262.301,Y 48.086,Z -10.000,A 0.015,B -0.000,C -180.000},{X -261.573,Y 46.547,Z -10.000,A 0.015,B 0.000,C -180.000} C_DIS
CIRC {X -260.881,Y 44.993,Z -10.000,A 0.015,B 0.000,C -180.000},{X -260.177,Y 43.444,Z -10.000,A 0.015,B 0.000,C 180.000} C_DIS
CIRC {X -257.629,Y 40.516,Z -10.000,A 0.015,B 0.000,C 180.000},{X -253.905,Y 39.425,Z -10.000,A 0.015,B 0.000,C 180.000} C_DIS
LIN {X -139.652,Y 39.425,Z -10.000,A 0.015,B -0.000,C -180.000} C_DIS
CIRC {X -135.892,Y 40.515,Z -10.000,A 0.015,B 0.000,C 180.000},{X -133.298,Y 43.448,Z -10.000,A 0.015,B 0.000,C -180.000} C_DIS
CIRC {X -132.491,Y 45.197,Z -10.000,A 0.015,B 0.000,C 180.000},{X -131.718,Y 46.960,Z -10.000,A 0.015,B 0.000,C 180.000} C_DIS
CIRC {X -130.908,Y 48.709,Z -10.000,A 0.015,B 0.000,C 180.000},{X -129.995,Y 50.405,Z -10.000,A 0.015,B -0.000,C -180.000} C_DIS
LIN {X -108.963,Y 86.155,Z -10.000,A 0.015,B -0.000,C 180.000} C_DIS
CIRC {X -96.188,Y 102.678,Z -10.000,A 0.015,B 0.000,C 180.000},{X -79.888,Y 115.736,Z -10.000,A 0.015,B 0.000,C -180.000} C_DIS
CIRC {X -76.151,Y 117.890,Z -10.000,A 0.015,B -0.000,C -180.000},{X -72.276,Y 119.783,Z -10.000,A 0.015,B 0.000,C 180.000} C_DIS
CIRC {X -68.350,Y 121.564,Z -10.000,A 0.015,B 0.000,C -180.000},{X -64.443,Y 123.386,Z -10.000,A 0.015,B -0.000,C -180.000} C_DIS
CIRC {X -61.510,Y 125.979,Z -10.000,A 0.015,B 0.000,C -180.000},{X -60.420,Y 129.738,Z -10.000,A 0.015,B 0.000,C -180.000} C_DIS
LIN {X -60.424,Y 264.664,Z -10.000,A 0.015,B 0.000,C 180.000} C_DIS
CIRC {X -61.552,Y 267.388,Z -10.000,A 0.015,B 0.000,C 180.000},{X -64.277,Y 268.516,Z -10.000,A 0.015,B 0.000,C -180.000} C_DIS
LIN {X -76.917,Y 268.516,Z -10.000,A 0.015,B 0.000,C 180.000} C_DIS
CIRC {X -80.308,Y 267.419,Z -10.000,A 0.015,B 0.000,C -180.000},{X -82.415,Y 264.545,Z -10.000,A 0.015,B 0.000,C -180.000} C_DIS
CIRC {X -91.293,Y 245.218,Z -10.000,A 0.015,B 0.000,C -180.000},{X -104.210,Y 228.321,Z -10.000,A 0.015,B 0.000,C 180.000} C_DIS
CIRC {X -120.357,Y 214.516,Z -10.000,A 0.015,B 0.000,C -180.000},{X -138.920,Y 204.187,Z -10.000,A 0.015,B 0.000,C -180.000} C_DIS
CIRC {X -157.313,Y 198.340,Z -10.000,A 0.015,B 0.000,C 180.000},{X -176.501,Y 196.269,Z -10.000,A 0.015,B 0.000,C -180.000} C_DIS
LIN {X -214.907,Y 196.131,Z -10.000,A 0.015,B 0.000,C 180.000} C_DIS
CIRC {X -233.029,Y 197.813,Z -10.000,A 0.015,B 0.000,C -180.000},{X -250.533,Y 202.798,Z -10.000,A 0.015,B 0.000,C 180.000} C_DIS
CIRC {X -266.909,Y 210.692,Z -10.000,A 0.015,B 0.000,C 180.000},{X -281.832,Y 221.076,Z -10.000,A 0.015,B 0.000,C 180.000} C_DIS
CIRC {X -286.056,Y 224.773,Z -10.000,A 0.015,B 0.000,C -180.000},{X -290.037,Y 228.730,Z -10.000,A 0.015,B 0.000,C 180.000} C_DIS
CIRC {X -292.051,Y 232.850,Z -10.000,A 0.015,B 0.000,C -180.000},{X -291.370,Y 237.385,Z -10.000,A 0.015,B 0.000,C -180.000} C_DIS
CIRC {X -290.504,Y 241.831,Z -10.000,A 0.015,B -0.000,C -180.000},{X -291.952,Y 246.123,Z -10.000,A 0.015,B 0.000,C 180.000} C_DIS
CIRC {X -292.807,Y 247.445,Z -10.000,A 0.015,B 0.000,C -180.000},{X -293.637,Y 248.784,Z -10.000,A 0.015,B 0.000,C 180.000} C_DIS
CIRC {X -299.766,Y 260.909,Z -10.000,A 0.015,B 0.000,C 180.000},{X -303.969,Y 273.829,Z -10.000,A 0.015,B 0.000,C -180.000} C_DIS
CIRC {X -305.840,Y 276.741,Z -10.000,A 0.015,B 0.000,C 180.000},{X -309.110,Y 277.873,Z -10.000,A 0.015,B 0.000,C 180.000} C_DIS
LIN {X -338.604,Y 277.872,Z -10.000,A 0.015,B -0.000,C -180.000} C_DIS
CIRC {X -341.329,Y 276.744,Z -10.000,A 0.015,B 0.000,C -180.000},{X -342.457,Y 274.019,Z -10.000,A 0.015,B 0.000,C -180.000} C_DIS
LIN {X -342.453,Y 123.091,Z -10.000,A 0.015,B 0.000,C -180.000} C_DIS
CIRC {X -341.364,Y 119.557,Z -10.000,A 0.015,B 0.000,C -180.000},{X -338.476,Y 117.250,Z -10.000,A 0.015,B 0.000,C 180.000} C_DIS
CIRC {X -329.763,Y 113.485,Z -10.000,A 0.015,B -0.000,C -180.000},{X -321.315,Y 109.158,Z -10.000,A 0.015,B 0.000,C -180.000} C_DIS
CIRC {X -313.323,Y 104.009,Z -10.000,A 0.015,B 0.000,C -180.000},{X -306.080,Y 97.851,Z -10.000,A 0.015,B 0.000,C 180.000} C_DIS
CIRC {X -295.492,Y 85.949,Z -10.000,A 0.015,B -0.000,C 180.000},{X -286.750,Y 72.633,Z -10.000,A 0.015,B 0.000,C 180.000} C_DIS
LIN {X -271.090,Y 44.986,Z -10.000,A 0.015,B 0.000,C -180.000} C_DIS
CIRC {X -269.723,Y 42.386,Z -10.000,A 0.015,B 0.000,C 180.000},{X -268.561,Y 39.689,Z -10.000,A 0.015,B 0.000,C 180.000} C_DIS
CIRC {X -267.520,Y 36.946,Z -10.000,A 0.015,B 0.000,C -180.000},{X -266.509,Y 34.191,Z -10.000,A 0.015,B 0.000,C -180.000} C_DIS
CIRC {X -264.222,Y 31.197,Z -10.000,A 0.015,B 0.000,C -180.000},{X -260.630,Y 30.062,Z -10.000,A 0.015,B 0.000,C 180.000} C_DIS
LIN {X -132.881,Y 30.062,Z -10.000,A 0.015,B 0.000,C 180.000} C_DIS
CIRC {X -129.339,Y 31.176,Z -10.000,A 0.015,B 0.000,C 180.000},{X -127.071,Y 34.116,Z -10.000,A 0.015,B 0.000,C -180.000} C_DIS
CIRC {X -122.336,Y 45.309,Z -10.000,A 0.015,B 0.000,C -180.000},{X -116.559,Y 56.002,Z -10.000,A 0.015,B 0.000,C 180.000} C_DIS
LIN {X -104.213,Y 76.909,Z -10.000,A 0.015,B 0.000,C 180.000} C_DIS
CIRC {X -98.151,Y 86.096,Z -10.000,A 0.015,B 0.000,C -180.000},{X -91.046,Y 94.502,Z -10.000,A 0.015,B 0.000,C -180.000} C_DIS
CIRC {X -82.965,Y 101.979,Z -10.000,A 0.015,B 0.000,C 180.000},{X -74.005,Y 108.377,Z -10.000,A 0.015,B 0.000,C -180.000} C_DIS
CIRC {X -69.460,Y 110.972,Z -10.000,A 0.015,B 0.000,C -180.000},{X -64.732,Y 113.214,Z -10.000,A 0.015,B -0.000,C 180.000} C_DIS
CIRC {X -59.911,Y 115.239,Z -10.000,A 0.015,B 0.000,C 180.000},{X -55.062,Y 117.197,Z -10.000,A 0.015,B 0.000,C 180.000} C_DIS
CIRC {X -52.153,Y 119.526,Z -10.000,A 0.015,B 0.000,C -180.000},{X -51.057,Y 123.088,Z -10.000,A 0.015,B 0.000,C 180.000} C_DIS
LIN {X -51.061,Y 274.026,Z -10.000,A 0.015,B 0.000,C -180.000} C_DIS
CIRC {X -52.190,Y 276.751,Z -10.000,A 0.015,B -0.000,C 180.000},{X -54.914,Y 277.879,Z -10.000,A 0.015,B 0.000,C 180.000} C_DIS
LIN {X -84.429,Y 277.879,Z -10.000,A 0.015,B 0.000,C -180.000} C_DIS
CIRC {X -87.691,Y 276.745,Z -10.000,A 0.015,B 0.000,C -180.000},{X -89.547,Y 273.834,Z -10.000,A 0.015,B 0.000,C 180.000} C_DIS
CIRC {X -96.736,Y 254.452,Z -10.000,A 0.015,B -0.000,C -180.000},{X -108.391,Y 237.379,Z -10.000,A 0.015,B 0.000,C 180.000} C_DIS
CIRC {X -123.646,Y 223.468,Z -10.000,A 0.015,B 0.000,C -180.000},{X -141.578,Y 213.238,Z -10.000,A 0.015,B -0.000,C 180.000} C_DIS
CIRC {X -160.065,Y 207.415,Z -10.000,A 0.015,B 0.000,C 180.000},{X -179.352,Y 205.488,Z -10.000,A 0.015,B 0.000,C -180.000} C_DIS
LIN {X -214.906,Y 205.493,Z -10.000,A 0.015,B 0.000,C 180.000} C_DIS
CIRC {X -231.427,Y 207.038,Z -10.000,A 0.015,B 0.000,C -180.000},{X -247.378,Y 211.613,Z -10.000,A 0.015,B -0.000,C -180.000} C_DIS
CIRC {X -262.294,Y 218.838,Z -10.000,A 0.015,B 0.000,C 180.000},{X -275.892,Y 228.313,Z -10.000,A 0.015,B 0.000,C -180.000} C_DIS
CIRC {X -284.590,Y 236.616,Z -10.000,A 0.015,B 0.000,C 180.000},{X -291.952,Y 246.123,Z -10.000,A 0.015,B -0.000,C 180.000} C_DIS
CIRC {X -293.256,Y 250.526,Z -10.000,A 0.015,B -0.000,C 180.000},{X -291.881,Y 254.907,Z -10.000,A 0.015,B 0.000,C 180.000} C_DIS
CIRC {X -290.363,Y 259.190,Z -10.000,A 0.015,B 0.000,C -180.000},{X -291.167,Y 263.663,Z -10.000,A 0.015,B -0.000,C 180.000} C_DIS
CIRC {X -292.908,Y 267.996,Z -10.000,A 0.015,B 0.000,C 180.000},{X -294.158,Y 272.495,Z -10.000,A 0.015,B 0.000,C 180.000} C_DIS
LIN {X -296.544,Y 283.206,Z -10.000,A 0.015,B -0.000,C -180.000} C_DIS
CIRC {X -298.360,Y 286.105,Z -10.000,A 0.015,B 0.000,C 180.000},{X -301.588,Y 287.236,Z -10.000,A 0.015,B 0.000,C 180.000} C_DIS
LIN {X -347.967,Y 287.235,Z -10.000,A 0.015,B 0.000,C 180.000} C_DIS
CIRC {X -350.692,Y 286.106,Z -10.000,A 0.015,B 0.000,C -180.000},{X -351.820,Y 283.382,Z -10.000,A 0.015,B 0.000,C -180.000} C_DIS
LIN {X -351.815,Y 115.597,Z -10.000,A 0.015,B 0.000,C -180.000} C_DIS
CIRC {X -350.727,Y 112.393,Z -10.000,A 0.015,B 0.000,C 180.000},{X -347.912,Y 110.515,Z -10.000,A 0.015,B 0.000,C -180.000} C_DIS
CIRC {X -333.546,Y 105.179,Z -10.000,A 0.015,B 0.000,C -180.000},{X -320.442,Y 97.233,Z -10.000,A 0.015,B 0.000,C 180.000} C_DIS
CIRC {X -308.960,Y 87.107,Z -10.000,A 0.015,B 0.000,C 180.000},{X -299.306,Y 75.226,Z -10.000,A 0.015,B 0.000,C -180.000} C_DIS
LIN {X -279.065,Y 40.390,Z -10.000,A 0.015,B 0.000,C -180.000} C_DIS
CIRC {X -277.173,Y 36.636,Z -10.000,A 0.015,B -0.000,C -180.000},{X -275.711,Y 32.694,Z -10.000,A 0.015,B 0.000,C -180.000} C_DIS
CIRC {X -274.426,Y 28.698,Z -10.000,A 0.015,B 0.000,C -180.000},{X -273.049,Y 24.733,Z -10.000,A 0.015,B 0.000,C 180.000} C_DIS
CIRC {X -270.816,Y 21.809,Z -10.000,A 0.015,B -0.000,C -180.000},{X -267.308,Y 20.700,Z -10.000,A 0.015,B 0.000,C 180.000} C_DIS
LIN {X -126.204,Y 20.700,Z -10.000,A 0.015,B 0.000,C 180.000} C_DIS
CIRC {X -122.671,Y 21.824,Z -10.000,A 0.015,B 0.000,C 180.000},{X -120.437,Y 24.784,Z -10.000,A 0.015,B 0.000,C 180.000} C_DIS
CIRC {X -119.001,Y 28.949,Z -10.000,A 0.015,B -0.000,C 180.000},{X -117.621,Y 33.133,Z -10.000,A 0.015,B 0.000,C -180.000} C_DIS
CIRC {X -116.046,Y 37.255,Z -10.000,A 0.015,B 0.000,C -180.000},{X -114.044,Y 41.187,Z -10.000,A 0.015,B 0.000,C -180.000} C_DIS
LIN {X -96.107,Y 72.224,Z -10.000,A 0.015,B 0.000,C 180.000} C_DIS
CIRC {X -86.599,Y 85.383,Z -10.000,A 0.015,B 0.000,C -180.000},{X -74.631,Y 96.352,Z -10.000,A 0.015,B 0.000,C 180.000} C_DIS
CIRC {X -60.777,Y 104.791,Z -10.000,A 0.015,B 0.000,C -180.000},{X -45.601,Y 110.518,Z -10.000,A 0.015,B 0.000,C 180.000} C_DIS
CIRC {X -42.782,Y 112.419,Z -10.000,A 0.015,B 0.000,C -180.000},{X -41.694,Y 115.640,Z -10.000,A 0.015,B 0.000,C 180.000} C_DIS
LIN {X -41.699,Y 283.389,Z -10.000,A 0.015,B 0.000,C -180.000} C_DIS
CIRC {X -42.828,Y 286.114,Z -10.000,A 0.015,B -0.000,C -180.000},{X -45.552,Y 287.242,Z -10.000,A 0.015,B -0.000,C 180.000} C_DIS
LIN {X -91.871,Y 287.241,Z -10.000,A 0.015,B 0.000,C 180.000} C_DIS
CIRC {X -95.099,Y 286.119,Z -10.000,A 0.015,B 0.000,C 180.000},{X -96.936,Y 283.238,Z -10.000,A 0.015,B -0.000,C -180.000} C_DIS
CIRC {X -98.401,Y 277.202,Z -10.000,A 0.015,B -0.000,C 180.000},{X -99.923,Y 271.181,Z -10.000,A 0.015,B 0.000,C -180.000} C_DIS
CIRC {X -101.835,Y 265.260,Z -10.000,A 0.015,B 0.000,C 180.000},{X -104.445,Y 259.612,Z -10.000,A 0.015,B -0.000,C 180.000} C_DIS
CIRC {X -109.025,Y 252.013,Z -10.000,A 0.015,B 0.000,C 180.000},{X -114.335,Y 244.905,Z -10.000,A 0.015,B 0.000,C -180.000} C_DIS
CIRC {X -120.397,Y 238.419,Z -10.000,A 0.015,B 0.000,C -180.000},{X -127.197,Y 232.712,Z -10.000,A 0.015,B 0.000,C 180.000} C_DIS
CIRC {X -133.760,Y 228.208,Z -10.000,A 0.015,B 0.000,C -180.000},{X -140.632,Y 224.191,Z -10.000,A 0.015,B 0.000,C 180.000} C_DIS
CIRC {X -147.857,Y 220.833,Z -10.000,A 0.015,B 0.000,C 180.000},{X -155.421,Y 218.328,Z -10.000,A 0.015,B -0.000,C 180.000} C_DIS
CIRC {X -170.107,Y 215.457,Z -10.000,A 0.015,B 0.000,C 180.000},{X -185.049,Y 214.638,Z -10.000,A 0.015,B 0.000,C -180.000} C_DIS
LIN {X -214.904,Y 214.856,Z -10.000,A 0.015,B 0.000,C 180.000} C_DIS
CIRC {X -229.826,Y 216.262,Z -10.000,A 0.015,B 0.000,C -180.000},{X -244.223,Y 220.428,Z -10.000,A 0.015,B 0.000,C -180.000} C_DIS
CIRC {X -257.678,Y 226.984,Z -10.000,A 0.015,B -0.000,C 180.000},{X -269.952,Y 235.550,Z -10.000,A 0.015,B 0.000,C 180.000} C_DIS
CIRC {X -276.139,Y 241.317,Z -10.000,A 0.015,B 0.000,C -180.000},{X -281.551,Y 247.816,Z -10.000,A 0.015,B 0.000,C -180.000} C_DIS
CIRC {X -286.270,Y 254.822,Z -10.000,A 0.015,B 0.000,C 180.000},{X -290.434,Y 262.171,Z -10.000,A 0.015,B 0.000,C 180.000} C_DIS
CIRC {X -290.808,Y 262.914,Z -10.000,A 0.015,B 0.000,C -180.000},{X -291.167,Y 263.663,Z -10.000,A 0.015,B -0.000,C 180.000} C_DIS
CIRC {X -291.782,Y 268.488,Z -10.000,A 0.015,B 0.000,C 180.000},{X -289.472,Y 272.769,Z -10.000,A 0.015,B 0.000,C 180.000} C_DIS
CIRC {X -286.987,Y 276.867,Z -10.000,A 0.015,B 0.000,C 180.000},{X -286.870,Y 281.658,Z -10.000,A 0.015,B 0.000,C 180.000} C_DIS
CIRC {X -288.023,Y 287.199,Z -10.000,A 0.015,B 0.000,C 180.000},{X -288.832,Y 292.801,Z -10.000,A 0.015,B 0.000,C -180.000} C_DIS
CIRC {X -290.234,Y 295.511,Z -10.000,A 0.015,B -0.000,C -180.000},{X -293.084,Y 296.599,Z -10.000,A 0.015,B 0.000,C -180.000} C_DIS
LIN {X -357.330,Y 296.597,Z -10.000,A 0.015,B 0.000,C 180.000} C_DIS
CIRC {X -360.055,Y 295.469,Z -10.000,A 0.015,B -0.000,C -180.000},{X -361.183,Y 292.744,Z -10.000,A 0.015,B 0.000,C 180.000} C_DIS
LIN {X -361.178,Y 107.286,Z -10.000,A 0.015,B 0.000,C -180.000} C_DIS
CIRC {X -360.087,Y 104.375,Z -10.000,A 0.015,B 0.000,C -180.000},{X -357.353,Y 102.897,Z -10.000,A 0.015,B 0.000,C 180.000} C_DIS
CIRC {X -348.814,Y 101.146,Z -10.000,A 0.015,B -0.000,C 180.000},{X -340.576,Y 98.299,Z -10.000,A 0.015,B 0.000,C 180.000} C_DIS
CIRC {X -332.747,Y 94.478,Z -10.000,A 0.015,B 0.000,C -180.000},{X -325.397,Y 89.802,Z -10.000,A 0.015,B 0.000,C 180.000} C_DIS
CIRC {X -320.112,Y 85.526,Z -10.000,A 0.015,B -0.000,C -180.000},{X -315.350,Y 80.674,Z -10.000,A 0.015,B 0.000,C 180.000} C_DIS
CIRC {X -311.033,Y 75.433,Z -10.000,A 0.015,B 0.000,C 180.000},{X -307.036,Y 69.943,Z -10.000,A 0.015,B 0.000,C 180.000} C_DIS
LIN {X -287.160,Y 35.725,Z -10.000,A 0.015,B 0.000,C -180.000} C_DIS
CIRC {X -284.699,Y 30.842,Z -10.000,A 0.015,B 0.000,C -180.000},{X -282.797,Y 25.716,Z -10.000,A 0.015,B 0.000,C 180.000} C_DIS
CIRC {X -281.250,Y 20.479,Z -10.000,A 0.015,B -0.000,C -180.000},{X -279.830,Y 15.207,Z -10.000,A 0.015,B 0.000,C 180.000} C_DIS
CIRC {X -277.999,Y 12.418,Z -10.000,A 0.015,B 0.000,C 180.000},{X -274.843,Y 11.337,Z -10.000,A 0.015,B -0.000,C 180.000} C_DIS
LIN {X -118.727,Y 11.337,Z -10.000,A 0.015,B -0.000,C 180.000} C_DIS
CIRC {X -115.531,Y 12.417,Z -10.000,A 0.015,B -0.000,C 180.000},{X -113.645,Y 15.214,Z -10.000,A 0.015,B 0.000,C -180.000} C_DIS
CIRC {X -108.912,Y 29.054,Z -10.000,A 0.015,B 0.000,C -180.000},{X -102.503,Y 42.200,Z -10.000,A 0.015,B 0.000,C -180.000} C_DIS
LIN {X -88.001,Y 67.539,Z -10.000,A 0.015,B 0.000,C -180.000} C_DIS
CIRC {X -66.106,Y 91.123,Z -10.000,A 0.015,B 0.000,C 180.000},{X -36.152,Y 102.883,Z -10.000,A 0.015,B -0.000,C -180.000} C_DIS
CIRC {X -33.417,Y 104.403,Z -10.000,A 0.015,B 0.000,C 180.000},{X -32.331,Y 107.337,Z -10.000,A 0.015,B -0.000,C 180.000} C_DIS
LIN {X -32.337,Y 292.752,Z -10.000,A 0.015,B -0.000,C 180.000} C_DIS
CIRC {X -33.465,Y 295.476,Z -10.000,A 0.015,B 0.000,C -180.000},{X -36.190,Y 296.605,Z -10.000,A 0.015,B -0.000,C -180.000} C_DIS
LIN {X -100.463,Y 296.603,Z -10.000,A 0.015,B 0.000,C -180.000} C_DIS
CIRC {X -103.297,Y 295.515,Z -10.000,A 0.015,B -0.000,C 180.000},{X -104.676,Y 292.810,Z -10.000,A 0.015,B -0.000,C 180.000} C_DIS
CIRC {X -105.721,Y 285.377,Z -10.000,A 0.015,B 0.000,C 180.000},{X -107.284,Y 278.035,Z -10.000,A 0.015,B 0.000,C -180.000} C_DIS
CIRC {X -109.554,Y 270.871,Z -10.000,A 0.015,B -0.000,C -180.000},{X -112.693,Y 264.042,Z -10.000,A 0.015,B 0.000,C -180.000} C_DIS
CIRC {X -116.737,Y 257.322,Z -10.000,A 0.015,B 0.000,C 180.000},{X -121.417,Y 251.029,Z -10.000,A 0.015,B 0.000,C 180.000} C_DIS
CIRC {X -126.764,Y 245.284,Z -10.000,A 0.015,B -0.000,C 180.000},{X -132.772,Y 240.234,Z -10.000,A 0.015,B 0.000,C 180.000} C_DIS
CIRC {X -138.605,Y 236.219,Z -10.000,A 0.015,B -0.000,C 180.000},{X -144.704,Y 232.621,Z -10.000,A 0.015,B 0.000,C 180.000} C_DIS
CIRC {X -151.121,Y 229.608,Z -10.000,A 0.015,B 0.000,C 180.000},{X -157.848,Y 227.370,Z -10.000,A 0.015,B 0.000,C 180.000} C_DIS
CIRC {X -171.938,Y 224.638,Z -10.000,A 0.015,B -0.000,C 180.000},{X -186.272,Y 223.920,Z -10.000,A 0.015,B -0.000,C 180.000} C_DIS
LIN {X -214.903,Y 224.219,Z -10.000,A 0.015,B -0.000,C -180.000} C_DIS
CIRC {X -228.224,Y 225.487,Z -10.000,A 0.015,B 0.000,C -180.000},{X -241.068,Y 229.243,Z -10.000,A 0.015,B -0.000,C -180.000} C_DIS
CIRC {X -253.062,Y 235.130,Z -10.000,A 0.015,B 0.000,C -180.000},{X -264.012,Y 242.787,Z -10.000,A 0.015,B 0.000,C 180.000} C_DIS
CIRC {X -273.962,Y 253.081,Z -10.000,A 0.015,B 0.000,C 180.000},{X -281.301,Y 265.373,Z -10.000,A 0.015,B -0.000,C -180.000} C_DIS
CIRC {X -284.467,Y 273.385,Z -10.000,A 0.015,B 0.000,C -180.000},{X -286.870,Y 281.658,Z -10.000,A 0.015,B 0.000,C 180.000} C_DIS
CIRC {X -286.564,Y 286.155,Z -10.000,A 0.015,B -0.000,C -180.000},{X -283.744,Y 289.673,Z -10.000,A 0.015,B 0.000,C 180.000} C_DIS
CIRC {X -280.777,Y 292.970,Z -10.000,A 0.015,B 0.000,C -180.000},{X -279.728,Y 297.280,Z -10.000,A 0.015,B -0.000,C 180.000} C_DIS
CIRC {X -279.686,Y 299.805,Z -10.000,A 0.015,B 0.000,C 180.000},{X -279.523,Y 302.324,Z -10.000,A 0.015,B 0.000,C -180.000} C_DIS
CIRC {X -280.385,Y 304.876,Z -10.000,A 0.015,B -0.000,C 180.000},{X -282.850,Y 305.962,Z -10.000,A 0.015,B 0.000,C 180.000} C_DIS
LIN {X -366.693,Y 305.960,Z -10.000,A 0.015,B 0.000,C 180.000} C_DIS
CIRC {X -369.417,Y 304.831,Z -10.000,A 0.015,B 0.000,C 180.000},{X -370.546,Y 302.107,Z -10.000,A 0.015,B 0.000,C -180.000} C_DIS
LIN {X -370.540,Y 98.688,Z -10.000,A 0.015,B 0.000,C 180.000} C_DIS
CIRC {X -369.422,Y 95.799,Z -10.000,A 0.015,B -0.000,C 180.000},{X -366.651,Y 94.414,Z -10.000,A 0.015,B 0.000,C -180.000} C_DIS
CIRC {X -361.840,Y 93.973,Z -10.000,A 0.015,B -0.000,C -180.000},{X -357.026,Y 93.561,Z -10.000,A 0.015,B 0.000,C 180.000} C_DIS
CIRC {X -352.243,Y 92.777,Z -10.000,A 0.015,B 0.000,C 180.000},{X -347.645,Y 91.243,Z -10.000,A 0.015,B 0.000,C -180.000} C_DIS
CIRC {X -337.464,Y 86.065,Z -10.000,A 0.015,B -0.000,C 180.000},{X -328.085,Y 79.547,Z -10.000,A 0.015,B 0.000,C 180.000} C_DIS
CIRC {X -319.860,Y 71.589,Z -10.000,A 0.015,B 0.000,C 180.000},{X -313.249,Y 62.247,Z -10.000,A 0.015,B 0.000,C 180.000} C_DIS
LIN {X -295.273,Y 31.051,Z -10.000,A 0.015,B 0.000,C -180.000} C_DIS
CIRC {X -292.312,Y 25.096,Z -10.000,A 0.015,B -0.000,C 180.000},{X -290.103,Y 18.825,Z -10.000,A 0.015,B 0.000,C -180.000} C_DIS
CIRC {X -288.578,Y 12.358,Z -10.000,A 0.015,B -0.000,C -180.000},{X -287.652,Y 5.779,Z -10.000,A 0.015,B 0.000,C -180.000} C_DIS
CIRC {X -286.298,Y 3.068,Z -10.000,A 0.015,B 0.000,C 180.000},{X -283.471,Y 1.974,Z -10.000,A 0.015,B 0.000,C 180.000} C_DIS
LIN {X -110.057,Y 1.974,Z -10.000,A 0.015,B 0.000,C 180.000} C_DIS
CIRC {X -107.226,Y 3.057,Z -10.000,A 0.015,B 0.000,C -180.000},{X -105.841,Y 5.753,Z -10.000,A 0.015,B -0.000,C -180.000} C_DIS
CIRC {X -104.803,Y 12.534,Z -10.000,A 0.015,B 0.000,C -180.000},{X -103.192,Y 19.202,Z -10.000,A 0.015,B 0.000,C -180.000} C_DIS
CIRC {X -100.898,Y 25.673,Z -10.000,A 0.015,B 0.000,C 180.000},{X -97.832,Y 31.817,Z -10.000,A 0.015,B 0.000,C -180.000} C_DIS
LIN {X -79.894,Y 62.854,Z -10.000,A 0.015,B 0.000,C -180.000} C_DIS
CIRC {X -73.144,Y 72.294,Z -10.000,A 0.015,B 0.000,C -180.000},{X -64.703,Y 80.258,Z -10.000,A 0.015,B 0.000,C -180.000} C_DIS
CIRC {X -55.074,Y 86.690,Z -10.000,A 0.015,B 0.000,C -180.000},{X -44.634,Y 91.700,Z -10.000,A 0.015,B 0.000,C -180.000} C_DIS
CIRC {X -40.316,Y 93.035,Z -10.000,A 0.015,B 0.000,C 180.000},{X -35.845,Y 93.695,Z -10.000,A 0.015,B 0.000,C -180.000} C_DIS
CIRC {X -31.351,Y 94.032,Z -10.000,A 0.015,B 0.000,C 180.000},{X -26.862,Y 94.419,Z -10.000,A 0.015,B 0.000,C -180.000} C_DIS
CIRC {X -24.088,Y 95.797,Z -10.000,A 0.015,B -0.000,C 180.000},{X -22.969,Y 98.684,Z -10.000,A 0.015,B 0.000,C 180.000} C_DIS
LIN {X -22.974,Y 302.115,Z -10.000,A 0.015,B -0.000,C -180.000} C_DIS
CIRC {X -24.103,Y 304.839,Z -10.000,A 0.015,B 0.000,C 180.000},{X -26.827,Y 305.968,Z -10.000,A 0.015,B 0.000,C -180.000} C_DIS
LIN {X -110.701,Y 305.966,Z -10.000,A 0.015,B 0.000,C 180.000} C_DIS
CIRC {X -113.148,Y 304.873,Z -10.000,A 0.015,B 0.000,C 180.000},{X -113.968,Y 302.322,Z -10.000,A 0.015,B 0.000,C -180.000} C_DIS
CIRC {X -113.721,Y 293.558,Z -10.000,A 0.015,B 0.000,C -180.000},{X -114.889,Y 284.868,Z -10.000,A 0.015,B -0.000,C -180.000} C_DIS
CIRC {X -117.343,Y 276.459,Z -10.000,A 0.015,B -0.000,C 180.000},{X -120.941,Y 268.472,Z -10.000,A 0.015,B 0.000,C 180.000} C_DIS
CIRC {X -124.449,Y 262.631,Z -10.000,A 0.015,B 0.000,C -180.000},{X -128.500,Y 257.152,Z -10.000,A 0.015,B -0.000,C 180.000} C_DIS
CIRC {X -133.131,Y 252.148,Z -10.000,A 0.015,B -0.000,C -180.000},{X -138.347,Y 247.756,Z -10.000,A 0.015,B 0.000,C 180.000} C_DIS
CIRC {X -143.450,Y 244.230,Z -10.000,A 0.015,B 0.000,C -180.000},{X -148.777,Y 241.052,Z -10.000,A 0.015,B 0.000,C 180.000} C_DIS
CIRC {X -154.385,Y 238.383,Z -10.000,A 0.015,B 0.000,C 180.000},{X -160.275,Y 236.413,Z -10.000,A 0.015,B 0.000,C 180.000} C_DIS
CIRC {X -173.769,Y 233.820,Z -10.000,A 0.015,B 0.000,C 180.000},{X -187.495,Y 233.203,Z -10.000,A 0.015,B 0.000,C -180.000} C_DIS
LIN {X -214.901,Y 233.581,Z -10.000,A 0.015,B 0.000,C -180.000} C_DIS
CIRC {X -226.623,Y 234.712,Z -10.000,A 0.015,B 0.000,C 180.000},{X -237.913,Y 238.058,Z -10.000,A 0.015,B 0.000,C 180.000} C_DIS
CIRC {X -248.447,Y 243.275,Z -10.000,A 0.015,B 0.000,C 180.000},{X -258.072,Y 250.024,Z -10.000,A 0.015,B 0.000,C -180.000} C_DIS
CIRC {X -265.045,Y 256.900,Z -10.000,A 0.015,B 0.000,C 180.000},{X -270.656,Y 264.927,Z -10.000,A 0.015,B 0.000,C -180.000} C_DIS
CIRC {X -274.897,Y 273.736,Z -10.000,A 0.015,B -0.000,C -180.000},{X -277.862,Y 283.052,Z -10.000,A 0.015,B 0.000,C -180.000} C_DIS
CIRC {X -278.839,Y 287.808,Z -10.000,A 0.015,B 0.000,C -180.000},{X -279.481,Y 292.620,Z -10.000,A 0.015,B -0.000,C -180.000} C_DIS
CIRC {X -279.657,Y 294.948,Z -10.000,A 0.015,B 0.000,C -180.000},{X -279.728,Y 297.280,Z -10.000,A 0.015,B 0.000,C 180.000} C_DIS
CIRC {X -278.373,Y 301.475,Z -10.000,A 0.015,B 0.000,C 180.000},{X -274.780,Y 304.029,Z -10.000,A 0.015,B 0.000,C 180.000} C_DIS
CIRC {X -271.128,Y 306.390,Z -10.000,A 0.015,B 0.000,C 180.000},{X -269.258,Y 310.317,Z -10.000,A 0.015,B 0.000,C 180.000} C_DIS
LIN {X -269.100,Y 311.297,Z -10.000,A 0.015,B 0.000,C 180.000} C_DIS
CIRC {X -269.835,Y 313.865,Z -10.000,A 0.015,B -0.000,C 180.000},{X -272.262,Y 314.980,Z -10.000,A 0.015,B 0.000,C -180.000} C_DIS
LIN {X -375.711,Y 314.977,Z -10.000,A 0.015,B -0.000,C -180.000} C_DIS
CIRC {X -378.436,Y 313.849,Z -10.000,A 0.015,B 0.000,C -180.000},{X -379.564,Y 311.124,Z -10.000,A 0.015,B 0.000,C -180.000} C_DIS
LIN {X -379.558,Y 88.798,Z -10.000,A 0.015,B 0.000,C -180.000} C_DIS
CIRC {X -378.483,Y 86.364,Z -10.000,A 0.015,B -0.000,C 180.000},{X -375.961,Y 85.517,Z -10.000,A 0.015,B 0.000,C -180.000} C_DIS
CIRC {X -365.445,Y 85.566,Z -10.000,A 0.015,B 0.000,C -180.000},{X -355.080,Y 83.792,Z -10.000,A 0.015,B -0.000,C -180.000} C_DIS
CIRC {X -345.190,Y 80.204,Z -10.000,A 0.015,B 0.000,C 180.000},{X -336.121,Y 74.873,Z -10.000,A 0.015,B 0.000,C -180.000} C_DIS
CIRC {X -332.093,Y 71.586,Z -10.000,A 0.015,B -0.000,C -180.000},{X -328.498,Y 67.830,Z -10.000,A 0.015,B 0.000,C -180.000} C_DIS
CIRC {X -325.249,Y 63.782,Z -10.000,A 0.015,B -0.000,C -180.000},{X -322.212,Y 59.573,Z -10.000,A 0.015,B 0.000,C 180.000} C_DIS
LIN {X -303.086,Y 26.548,Z -10.000,A 0.015,B 0.000,C -180.000} C_DIS
CIRC {X -300.407,Y 21.159,Z -10.000,A 0.015,B 0.000,C 180.000},{X -298.409,Y 15.483,Z -10.000,A 0.015,B -0.000,C -180.000} C_DIS
CIRC {X -297.060,Y 9.621,Z -10.000,A 0.015,B 0.000,C -180.000},{X -296.315,Y 3.653,Z -10.000,A 0.015,B 0.000,C 180.000} C_DIS
CIRC {X -296.268,Y 1.928,Z -10.000,A 0.015,B 0.000,C 180.000},{X -296.380,Y 0.205,Z -10.000,A 0.015,B 0.000,C 180.000} C_DIS
CIRC {X -296.545,Y -1.512,Z -10.000,A 0.015,B -0.000,C -180.000},{X -296.655,Y -3.233,Z -10.000,A 0.015,B 0.000,C 180.000} C_DIS
CIRC {X -295.654,Y -5.916,Z -10.000,A 0.015,B 0.000,C -180.000},{X -293.022,Y -7.044,Z -10.000,A 0.015,B 0.000,C 180.000} C_DIS
LIN {X -100.490,Y -7.044,Z -10.000,A 0.015,B 0.000,C 180.000} C_DIS
CIRC {X -97.858,Y -5.916,Z -10.000,A 0.015,B -0.000,C 180.000},{X -96.857,Y -3.233,Z -10.000,A 0.015,B 0.000,C 180.000} C_DIS
CIRC {X -97.009,Y 0.208,Z -10.000,A 0.015,B 0.000,C -180.000},{X -97.134,Y 3.651,Z -10.000,A 0.015,B 0.000,C 180.000} C_DIS
CIRC {X -96.987,Y 7.102,Z -10.000,A 0.015,B -0.000,C 180.000},{X -96.324,Y 10.492,Z -10.000,A 0.015,B 0.000,C -180.000} C_DIS
CIRC {X -95.075,Y 14.813,Z -10.000,A 0.015,B 0.000,C -180.000},{X -93.712,Y 19.100,Z -10.000,A 0.015,B 0.000,C 180.000} C_DIS
CIRC {X -92.076,Y 23.296,Z -10.000,A 0.015,B -0.000,C -180.000},{X -90.024,Y 27.305,Z -10.000,A 0.015,B 0.000,C 180.000} C_DIS
LIN {X -72.087,Y 58.342,Z -10.000,A 0.015,B 0.000,C 180.000} C_DIS
CIRC {X -66.197,Y 66.543,Z -10.000,A 0.015,B 0.000,C -180.000},{X -58.813,Y 73.430,Z -10.000,A 0.015,B 0.000,C -180.000} C_DIS
CIRC {X -50.405,Y 78.975,Z -10.000,A 0.015,B 0.000,C -180.000},{X -41.317,Y 83.314,Z -10.000,A 0.015,B 0.000,C -180.000} C_DIS
CIRC {X -35.544,Y 85.057,Z -10.000,A 0.015,B -0.000,C 180.000},{X -29.562,Y 85.814,Z -10.000,A 0.015,B -0.000,C 180.000} C_DIS
CIRC {X -23.549,Y 85.867,Z -10.000,A 0.015,B 0.000,C -180.000},{X -17.547,Y 85.517,Z -10.000,A 0.015,B 0.000,C 180.000} C_DIS
CIRC {X -15.025,Y 86.363,Z -10.000,A 0.015,B -0.000,C 180.000},{X -13.950,Y 88.798,Z -10.000,A 0.015,B 0.000,C 180.000} C_DIS
LIN {X -13.957,Y 311.133,Z -10.000,A 0.015,B 0.000,C -180.000} C_DIS
CIRC {X -15.085,Y 313.857,Z -10.000,A 0.015,B -0.000,C 180.000},{X -17.810,Y 314.986,Z -10.000,A 0.015,B 0.000,C 180.000} C_DIS
LIN {X -121.247,Y 314.983,Z -10.000,A 0.015,B 0.000,C 180.000} C_DIS
CIRC {X -123.657,Y 313.880,Z -10.000,A 0.015,B 0.000,C 180.000},{X -124.394,Y 311.335,Z -10.000,A 0.015,B 0.000,C 180.000} C_DIS
CIRC {X -123.608,Y 306.305,Z -10.000,A 0.015,B -0.000,C 180.000},{X -122.744,Y 301.288,Z -10.000,A 0.015,B 0.000,C -180.000} C_DIS
CIRC {X -122.359,Y 296.184,Z -10.000,A 0.015,B 0.000,C -180.000},{X -123.024,Y 291.110,Z -10.000,A 0.015,B -0.000,C -180.000} C_DIS
CIRC {X -124.391,Y 285.566,Z -10.000,A 0.015,B 0.000,C 180.000},{X -125.855,Y 280.048,Z -10.000,A 0.015,B 0.000,C -180.000} C_DIS
CIRC {X -127.850,Y 274.675,Z -10.000,A 0.015,B 0.000,C 180.000},{X -130.752,Y 269.733,Z -10.000,A 0.015,B 0.000,C -180.000} C_DIS
CIRC {X -137.546,Y 261.347,Z -10.000,A 0.015,B -0.000,C 180.000},{X -145.327,Y 253.868,Z -10.000,A 0.015,B -0.000,C -180.000} C_DIS
CIRC {X -154.453,Y 247.976,Z -10.000,A 0.015,B 0.000,C 180.000},{X -164.789,Y 244.630,Z -10.000,A 0.015,B 0.000,C -180.000} C_DIS
LIN {X -172.308,Y 243.239,Z -10.000,A 0.015,B 0.000,C -180.000} C_DIS
CIRC {X -175.812,Y 242.755,Z -10.000,A 0.015,B 0.000,C 180.000},{X -179.347,Y 242.594,Z -10.000,A 0.015,B -0.000,C -180.000} C_DIS
LIN {X -214.900,Y 242.599,Z -10.000,A 0.015,B -0.000,C 180.000} C_DIS
CIRC {X -225.080,Y 243.597,Z -10.000,A 0.015,B 0.000,C 180.000},{X -234.874,Y 246.548,Z -10.000,A 0.015,B 0.000,C -180.000} C_DIS
CIRC {X -244.001,Y 251.121,Z -10.000,A 0.015,B 0.000,C 180.000},{X -252.351,Y 256.995,Z -10.000,A 0.015,B -0.000,C -180.000} C_DIS
CIRC {X -258.278,Y 262.861,Z -10.000,A 0.015,B 0.000,C -180.000},{X -263.019,Y 269.722,Z -10.000,A 0.015,B 0.000,C -180.000} C_DIS
CIRC {X -266.588,Y 277.240,Z -10.000,A 0.015,B 0.000,C 180.000},{X -269.097,Y 285.176,Z -10.000,A 0.015,B 0.000,C -180.000} C_DIS
CIRC {X -269.967,Y 289.194,Z -10.000,A 0.015,B 0.000,C 180.000},{X -270.639,Y 293.249,Z -10.000,A 0.015,B 0.000,C 180.000} C_DIS
CIRC {X -270.980,Y 297.351,Z -10.000,A 0.015,B 0.000,C 180.000},{X -270.858,Y 301.465,Z -10.000,A 0.015,B 0.000,C 180.000} C_DIS
CIRC {X -270.551,Y 303.945,Z -10.000,A 0.015,B 0.000,C 180.000},{X -270.060,Y 306.395,Z -10.000,A 0.015,B 0.000,C -180.000} C_DIS
CIRC {X -269.626,Y 308.349,Z -10.000,A 0.015,B 0.000,C -180.000},{X -269.258,Y 310.317,Z -10.000,A 0.015,B 0.000,C 180.000} C_DIS
CIRC {X -267.757,Y 313.874,Z -10.000,A 0.015,B -0.000,C 180.000},{X -264.827,Y 316.390,Z -10.000,A 0.015,B -0.000,C -180.000} C_DIS
CIRC {X -262.850,Y 320.742,Z -10.000,A 0.015,B 0.000,C -180.000},{X -266.609,Y 323.694,Z -10.000,A 0.015,B 0.000,C -180.000} C_DIS
LIN {X -384.425,Y 323.691,Z -10.000,A 0.015,B -0.000,C -180.000} C_DIS
CIRC {X -387.150,Y 322.562,Z -10.000,A 0.015,B 0.000,C -180.000},{X -388.278,Y 319.838,Z -10.000,A 0.015,B -0.000,C -180.000} C_DIS
LIN {X -388.271,Y 77.065,Z -10.000,A 0.015,B 0.000,C -180.000} C_DIS
CIRC {X -387.149,Y 74.829,Z -10.000,A 0.015,B 0.000,C -180.000},{X -384.686,Y 74.391,Z -10.000,A 0.015,B 0.000,C 180.000} C_DIS
CIRC {X -381.033,Y 75.486,Z -10.000,A 0.015,B 0.000,C 180.000},{X -377.385,Y 76.599,Z -10.000,A 0.015,B -0.000,C -180.000} C_DIS
CIRC {X -373.630,Y 77.361,Z -10.000,A 0.015,B 0.000,C -180.000},{X -369.798,Y 77.376,Z -10.000,A 0.015,B -0.000,C -180.000} C_DIS
CIRC {X -360.777,Y 76.034,Z -10.000,A 0.015,B -0.000,C 180.000},{X -351.951,Y 73.738,Z -10.000,A 0.015,B 0.000,C -180.000} C_DIS
CIRC {X -343.657,Y 69.765,Z -10.000,A 0.015,B 0.000,C 180.000},{X -336.771,Y 63.670,Z -10.000,A 0.015,B 0.000,C -180.000} C_DIS
CIRC {X -334.625,Y 61.185,Z -10.000,A 0.015,B -0.000,C -180.000},{X -332.455,Y 58.721,Z -10.000,A 0.015,B 0.000,C -180.000} C_DIS
CIRC {X -330.398,Y 56.155,Z -10.000,A 0.015,B -0.000,C 180.000},{X -328.613,Y 53.394,Z -10.000,A 0.015,B 0.000,C -180.000} C_DIS
LIN {X -310.636,Y 22.198,Z -10.000,A 0.015,B 0.000,C -180.000} C_DIS
CIRC {X -307.031,Y 14.064,Z -10.000,A 0.015,B 0.000,C -180.000},{X -305.209,Y 5.356,Z -10.000,A 0.015,B 0.000,C 180.000} C_DIS
CIRC {X -305.027,Y -3.518,Z -10.000,A 0.015,B 0.000,C 180.000},{X -306.264,Y -12.307,Z -10.000,A 0.015,B 0.000,C -180.000} C_DIS
CIRC {X -305.711,Y -14.696,Z -10.000,A 0.015,B 0.000,C -180.000},{X -303.500,Y -15.758,Z -10.000,A 0.015,B 0.000,C 180.000} C_DIS
LIN {X -89.976,Y -15.758,Z -10.000,A 0.015,B -0.000,C 180.000} C_DIS
CIRC {X -87.766,Y -14.684,Z -10.000,A 0.015,B 0.000,C 180.000},{X -87.245,Y -12.282,Z -10.000,A 0.015,B 0.000,C 180.000} C_DIS
CIRC {X -88.500,Y -3.695,Z -10.000,A 0.015,B 0.000,C -180.000},{X -88.138,Y 4.977,Z -10.000,A 0.015,B 0.000,C 180.000} C_DIS
CIRC {X -86.314,Y 13.450,Z -10.000,A 0.015,B 0.000,C -180.000},{X -83.214,Y 21.544,Z -10.000,A 0.015,B -0.000,C 180.000} C_DIS
LIN {X -64.542,Y 53.982,Z -10.000,A 0.015,B 0.000,C 180.000} C_DIS
CIRC {X -59.485,Y 60.987,Z -10.000,A 0.015,B 0.000,C 180.000},{X -53.121,Y 66.831,Z -10.000,A 0.015,B 0.000,C -180.000} C_DIS
CIRC {X -45.894,Y 71.519,Z -10.000,A 0.015,B 0.000,C 180.000},{X -38.111,Y 75.212,Z -10.000,A 0.015,B 0.000,C -180.000} C_DIS
CIRC {X -33.553,Y 76.592,Z -10.000,A 0.015,B 0.000,C 180.000},{X -28.831,Y 77.205,Z -10.000,A 0.015,B -0.000,C 180.000} C_DIS
CIRC {X -24.086,Y 77.325,Z -10.000,A 0.015,B 0.000,C -180.000},{X -19.340,Y 77.244,Z -10.000,A 0.015,B 0.000,C -180.000} C_DIS
CIRC {X -16.618,Y 76.913,Z -10.000,A 0.015,B -0.000,C 180.000},{X -13.987,Y 76.140,Z -10.000,A 0.015,B 0.000,C -180.000} C_DIS
CIRC {X -11.420,Y 75.204,Z -10.000,A 0.015,B 0.000,C 180.000},{X -8.818,Y 74.367,Z -10.000,A 0.015,B 0.000,C 180.000} C_DIS
CIRC {X -6.358,Y 74.797,Z -10.000,A 0.015,B 0.000,C 180.000},{X -5.236,Y 77.029,Z -10.000,A 0.015,B 0.000,C -180.000} C_DIS
LIN {X -5.243,Y 319.847,Z -10.000,A 0.015,B -0.000,C 180.000} C_DIS
CIRC {X -6.371,Y 322.572,Z -10.000,A 0.015,B 0.000,C -180.000},{X -9.096,Y 323.700,Z -10.000,A 0.015,B -0.000,C -180.000} C_DIS
LIN {X -134.692,Y 323.697,Z -10.000,A 0.015,B 0.000,C -180.000} C_DIS
CIRC {X -136.658,Y 322.580,Z -10.000,A 0.015,B -0.000,C 180.000},{X -136.704,Y 320.320,Z -10.000,A 0.015,B 0.000,C -180.000} C_DIS
CIRC {X -135.511,Y 318.073,Z -10.000,A 0.015,B 0.000,C 180.000},{X -134.356,Y 315.806,Z -10.000,A 0.015,B 0.000,C -180.000} C_DIS
CIRC {X -133.400,Y 313.440,Z -10.000,A 0.015,B 0.000,C 180.000},{X -132.828,Y 310.953,Z -10.000,A 0.015,B 0.000,C -180.000} C_DIS
CIRC {X -132.120,Y 306.519,Z -10.000,A 0.015,B 0.000,C 180.000},{X -131.314,Y 302.102,Z -10.000,A 0.015,B 0.000,C 180.000} C_DIS
CIRC {X -130.930,Y 297.603,Z -10.000,A 0.015,B -0.000,C -180.000},{X -131.502,Y 293.123,Z -10.000,A 0.015,B 0.000,C 180.000} C_DIS
LIN {X -133.790,Y 283.648,Z -10.000,A 0.015,B 0.000,C -180.000} C_DIS
CIRC {X -135.401,Y 279.025,Z -10.000,A 0.015,B 0.000,C -180.000},{X -137.851,Y 274.787,Z -10.000,A 0.015,B -0.000,C -180.000} C_DIS
CIRC {X -143.551,Y 267.661,Z -10.000,A 0.015,B -0.000,C 180.000},{X -150.011,Y 261.216,Z -10.000,A 0.015,B -0.000,C 180.000} C_DIS
CIRC {X -157.643,Y 256.085,Z -10.000,A 0.015,B 0.000,C 180.000},{X -166.374,Y 253.198,Z -10.000,A 0.015,B 0.000,C -180.000} C_DIS
CIRC {X -169.598,Y 252.589,Z -10.000,A 0.015,B 0.000,C -180.000},{X -172.816,Y 251.956,Z -10.000,A 0.015,B 0.000,C 180.000} C_DIS
CIRC {X -176.065,Y 251.470,Z -10.000,A 0.015,B 0.000,C -180.000},{X -179.345,Y 251.307,Z -10.000,A 0.015,B -0.000,C 180.000} C_DIS
LIN {X -214.898,Y 251.313,Z -10.000,A 0.015,B 0.000,C -180.000} C_DIS
CIRC {X -223.590,Y 252.182,Z -10.000,A 0.015,B -0.000,C 180.000},{X -231.937,Y 254.752,Z -10.000,A 0.015,B 0.000,C 180.000} C_DIS
CIRC {X -239.705,Y 258.703,Z -10.000,A 0.015,B -0.000,C -180.000},{X -246.822,Y 263.730,Z -10.000,A 0.015,B 0.000,C 180.000} C_DIS
CIRC {X -251.739,Y 268.621,Z -10.000,A 0.015,B 0.000,C 180.000},{X -255.639,Y 274.355,Z -10.000,A 0.015,B 0.000,C 180.000} C_DIS
CIRC {X -258.559,Y 280.626,Z -10.000,A 0.015,B 0.000,C 180.000},{X -260.629,Y 287.228,Z -10.000,A 0.015,B 0.000,C 180.000} C_DIS
CIRC {X -261.885,Y 294.875,Z -10.000,A 0.015,B 0.000,C -180.000},{X -261.985,Y 302.623,Z -10.000,A 0.015,B 0.000,C -180.000} C_DIS
CIRC {X -260.820,Y 310.293,Z -10.000,A 0.015,B 0.000,C 180.000},{X -258.319,Y 317.637,Z -10.000,A 0.015,B 0.000,C -180.000} C_DIS
CIRC {X -257.983,Y 318.328,Z -10.000,A 0.015,B -0.000,C -180.000},{X -257.599,Y 318.993,Z -10.000,A 0.015,B 0.000,C -180.000} C_DIS
CIRC {X -257.201,Y 319.650,Z -10.000,A 0.015,B 0.000,C -180.000},{X -256.824,Y 320.319,Z -10.000,A 0.015,B 0.000,C -180.000} C_DIS
CIRC {X -256.868,Y 322.577,Z -10.000,A 0.015,B 0.000,C -180.000},{X -258.832,Y 323.694,Z -10.000,A 0.015,B 0.000,C -180.000} C_DIS
LIN {X -266.609,Y 323.694,Z -10.000,A 0.015,B -0.000,C 180.000} C_DIS
CIRC {X -270.283,Y 324.806,Z -10.000,A 0.015,B 0.000,C -180.000},{X -272.722,Y 327.769,Z -10.000,A 0.015,B 0.000,C 180.000} C_DIS
CIRC {X -275.161,Y 330.731,Z -10.000,A 0.015,B 0.000,C 180.000},{X -278.834,Y 331.843,Z -10.000,A 0.015,B 0.000,C 180.000} C_DIS
LIN {X -392.575,Y 331.840,Z -10.000,A 0.015,B -0.000,C 180.000} C_DIS
CIRC {X -395.300,Y 330.712,Z -10.000,A 0.015,B 0.000,C 180.000},{X -396.428,Y 327.987,Z -10.000,A 0.015,B 0.000,C 180.000} C_DIS
LIN {X -396.421,Y 62.529,Z -10.000,A 0.015,B 0.000,C -180.000} C_DIS
CIRC {X -395.309,Y 60.755,Z -10.000,A 0.015,B 0.000,C 180.000},{X -393.227,Y 60.983,Z -10.000,A 0.015,B 0.000,C 180.000} C_DIS
CIRC {X -391.472,Y 62.377,Z -10.000,A 0.015,B 0.000,C 180.000},{X -389.723,Y 63.778,Z -10.000,A 0.015,B 0.000,C -180.000} C_DIS
CIRC {X -387.840,Y 65.013,Z -10.000,A 0.015,B -0.000,C -180.000},{X -385.754,Y 65.861,Z -10.000,A 0.015,B -0.000,C -180.000} C_DIS
CIRC {X -382.019,Y 67.035,Z -10.000,A 0.015,B -0.000,C -180.000},{X -378.323,Y 68.326,Z -10.000,A 0.015,B 0.000,C 180.000} C_DIS
CIRC {X -374.497,Y 69.264,Z -10.000,A 0.015,B -0.000,C 180.000},{X -370.558,Y 69.332,Z -10.000,A 0.015,B -0.000,C -180.000} C_DIS
CIRC {X -363.063,Y 68.275,Z -10.000,A 0.015,B 0.000,C -180.000},{X -355.695,Y 66.539,Z -10.000,A 0.015,B 0.000,C 180.000} C_DIS
CIRC {X -348.728,Y 63.395,Z -10.000,A 0.015,B 0.000,C -180.000},{X -342.965,Y 58.374,Z -10.000,A 0.015,B -0.000,C 180.000} C_DIS
CIRC {X -341.056,Y 56.179,Z -10.000,A 0.015,B -0.000,C 180.000},{X -339.110,Y 54.018,Z -10.000,A 0.015,B 0.000,C 180.000} C_DIS
CIRC {X -337.264,Y 51.765,Z -10.000,A 0.015,B 0.000,C 180.000},{X -335.674,Y 49.325,Z -10.000,A 0.015,B 0.000,C -180.000} C_DIS
LIN {X -317.697,Y 18.129,Z -10.000,A 0.015,B 0.000,C 180.000} C_DIS
CIRC {X -314.842,Y 11.627,Z -10.000,A 0.015,B 0.000,C 180.000},{X -313.460,Y 4.661,Z -10.000,A 0.015,B 0.000,C 180.000} C_DIS
CIRC {X -313.202,Y -2.402,Z -10.000,A 0.015,B 0.000,C 180.000},{X -313.657,Y -9.455,Z -10.000,A 0.015,B 0.000,C -180.000} C_DIS
CIRC {X -314.323,Y -12.426,Z -10.000,A 0.015,B 0.000,C 180.000},{X -315.598,Y -15.190,Z -10.000,A 0.015,B 0.000,C 180.000} C_DIS
CIRC {X -317.081,Y -17.830,Z -10.000,A 0.015,B -0.000,C -180.000},{X -318.428,Y -20.543,Z -10.000,A 0.015,B 0.000,C -180.000} C_DIS
CIRC {X -318.277,Y -22.813,Z -10.000,A 0.015,B -0.000,C -180.000},{X -316.281,Y -23.907,Z -10.000,A 0.015,B 0.000,C 180.000} C_DIS
LIN {X -77.202,Y -23.907,Z -10.000,A 0.015,B 0.000,C -180.000} C_DIS
CIRC {X -75.219,Y -22.806,Z -10.000,A 0.015,B 0.000,C 180.000},{X -75.106,Y -20.541,Z -10.000,A 0.015,B 0.000,C -180.000} C_DIS
CIRC {X -76.719,Y -17.218,Z -10.000,A 0.015,B -0.000,C 180.000},{X -78.297,Y -13.877,Z -10.000,A 0.015,B 0.000,C -180.000} C_DIS
CIRC {X -79.575,Y -10.397,Z -10.000,A 0.015,B 0.000,C 180.000},{X -80.251,Y -6.753,Z -10.000,A 0.015,B 0.000,C 180.000} C_DIS
CIRC {X -80.533,Y -3.182,Z -10.000,A 0.015,B 0.000,C 180.000},{X -80.670,Y 0.398,Z -10.000,A 0.015,B -0.000,C 180.000} C_DIS
CIRC {X -80.477,Y 3.983,Z -10.000,A 0.015,B 0.000,C 180.000},{X -79.776,Y 7.505,Z -10.000,A 0.015,B 0.000,C 180.000} C_DIS
CIRC {X -78.045,Y 12.865,Z -10.000,A 0.015,B 0.000,C -180.000},{X -75.850,Y 18.053,Z -10.000,A 0.015,B 0.000,C -180.000} C_DIS
LIN {X -57.486,Y 49.904,Z -10.000,A 0.015,B 0.000,C 180.000} C_DIS
CIRC {X -53.206,Y 55.790,Z -10.000,A 0.015,B 0.000,C 180.000},{X -47.798,Y 60.660,Z -10.000,A 0.015,B 0.000,C 180.000} C_DIS
CIRC {X -41.675,Y 64.547,Z -10.000,A 0.015,B -0.000,C 180.000},{X -35.113,Y 67.633,Z -10.000,A 0.015,B 0.000,C -180.000} C_DIS
CIRC {X -31.357,Y 68.771,Z -10.000,A 0.015,B -0.000,C 180.000},{X -27.466,Y 69.274,Z -10.000,A 0.015,B 0.000,C 180.000} C_DIS
CIRC {X -23.556,Y 69.371,Z -10.000,A 0.015,B 0.000,C 180.000},{X -19.645,Y 69.304,Z -10.000,A 0.015,B 0.000,C 180.000} C_DIS
CIRC {X -15.485,Y 68.804,Z -10.000,A 0.015,B 0.000,C -180.000},{X -11.461,Y 67.640,Z -10.000,A 0.015,B 0.000,C -180.000} C_DIS
CIRC {X -7.623,Y 65.984,Z -10.000,A 0.015,B 0.000,C -180.000},{X -3.948,Y 63.992,Z -10.000,A 0.015,B 0.000,C 180.000} C_DIS
CIRC {X -2.963,Y 63.323,Z -10.000,A 0.015,B 0.000,C -180.000},{X -2.059,Y 62.548,Z -10.000,A 0.015,B 0.000,C 180.000} C_DIS
CIRC {X -1.182,Y 61.744,Z -10.000,A 0.015,B 0.000,C 180.000},{X -0.272,Y 60.979,Z -10.000,A 0.015,B 0.000,C 180.000} C_DIS
CIRC {X 1.802,Y 60.741,Z -10.000,A 0.015,B 0.000,C -180.000},{X 2.914,Y 62.507,Z -10.000,A 0.015,B 0.000,C 180.000} C_DIS
LIN {X 2.907,Y 327.997,Z -10.000,A 0.015,B 0.000,C -180.000} C_DIS
CIRC {X 1.778,Y 330.722,Z -10.000,A 0.015,B 0.000,C 180.000},{X -0.946,Y 331.850,Z -10.000,A 0.015,B 0.000,C -180.000} C_DIS
LIN {X -150.158,Y 331.846,Z -10.000,A 0.015,B -0.000,C 180.000} C_DIS
CIRC {X -151.804,Y 330.738,Z -10.000,A 0.015,B 0.000,C 180.000},{X -151.395,Y 328.796,Z -10.000,A 0.015,B 0.000,C 180.000} C_DIS
CIRC {X -145.416,Y 321.357,Z -10.000,A 0.015,B -0.000,C 180.000},{X -141.436,Y 312.682,Z -10.000,A 0.015,B -0.000,C 180.000} C_DIS
CIRC {X -140.194,Y 308.366,Z -10.000,A 0.015,B -0.000,C 180.000},{X -139.222,Y 303.982,Z -10.000,A 0.015,B 0.000,C -180.000} C_DIS
CIRC {X -138.854,Y 299.483,Z -10.000,A 0.015,B 0.000,C -180.000},{X -139.431,Y 295.007,Z -10.000,A 0.015,B -0.000,C 180.000} C_DIS
CIRC {X -141.367,Y 287.936,Z -10.000,A 0.015,B -0.000,C -180.000},{X -143.781,Y 281.014,Z -10.000,A 0.015,B 0.000,C -180.000} C_DIS
CIRC {X -147.397,Y 274.557,Z -10.000,A 0.015,B 0.000,C 180.000},{X -152.665,Y 269.359,Z -10.000,A 0.015,B 0.000,C 180.000} C_DIS
CIRC {X -158.718,Y 265.425,Z -10.000,A 0.015,B 0.000,C -180.000},{X -165.208,Y 262.262,Z -10.000,A 0.015,B 0.000,C -180.000} C_DIS
CIRC {X -172.138,Y 260.165,Z -10.000,A 0.015,B 0.000,C 180.000},{X -179.344,Y 259.457,Z -10.000,A 0.015,B 0.000,C 180.000} C_DIS
LIN {X -214.897,Y 259.463,Z -10.000,A 0.015,B 0.000,C -180.000} C_DIS
CIRC {X -222.196,Y 260.212,Z -10.000,A 0.015,B -0.000,C 180.000},{X -229.191,Y 262.425,Z -10.000,A 0.015,B 0.000,C 180.000} C_DIS
CIRC {X -235.687,Y 265.793,Z -10.000,A 0.015,B -0.000,C 180.000},{X -241.652,Y 270.030,Z -10.000,A 0.015,B -0.000,C 180.000} C_DIS
CIRC {X -245.623,Y 274.008,Z -10.000,A 0.015,B 0.000,C 180.000},{X -248.737,Y 278.688,Z -10.000,A 0.015,B -0.000,C -180.000} C_DIS
CIRC {X -251.050,Y 283.793,Z -10.000,A 0.015,B 0.000,C 180.000},{X -252.708,Y 289.147,Z -10.000,A 0.015,B -0.000,C 180.000} C_DIS
CIRC {X -253.974,Y 299.767,Z -10.000,A 0.015,B -0.000,C 180.000},{X -252.698,Y 310.386,Z -10.000,A 0.015,B 0.000,C 180.000} C_DIS
CIRC {X -248.717,Y 320.347,Z -10.000,A 0.015,B -0.000,C -180.000},{X -242.112,Y 328.799,Z -10.000,A 0.015,B 0.000,C 180.000} C_DIS
CIRC {X -241.698,Y 330.736,Z -10.000,A 0.015,B 0.000,C 180.000},{X -243.339,Y 331.844,Z -10.000,A 0.015,B 0.000,C -180.000} C_DIS
LIN {X -278.834,Y 331.843,Z -10.000,A 0.015,B 0.000,C -180.000} C_DIS
LIN {X -279.443,Y 331.688,Z -9.830,A 0.015,B 0.000,C 180.000} C_DIS
LIN {X -279.802,Y 331.396,Z -9.365,A 0.015,B 0.000,C 180.000} C_DIS
LIN {X -279.903,Y 331.259,Z -8.730,A 0.015,B 0.000,C 180.000} C_DIS
$VEL.CP = 1.00000
LIN {X -279.903,Y 331.259,Z 11.769,A 0.015,B 0.000,C -180.000} C_DIS
$VEL.CP = 1.00000
LIN {X -398.503,Y 339.199,Z 11.769,A 0.015,B 0.000,C -180.000} C_DIS
$VEL.CP = 0.10000
LIN {X -398.507,Y 339.199,Z 11.679,A 0.015,B -0.000,C 180.000} C_DIS
LIN {X -398.632,Y 339.197,Z 11.212,A 0.015,B 0.000,C -180.000} C_DIS
LIN {X -398.924,Y 339.182,Z 10.825,A 0.015,B -0.000,C -180.000} C_DIS
LIN {X -399.336,Y 339.133,Z 10.576,A 0.015,B -0.000,C 180.000} C_DIS
LIN {X -399.692,Y 339.076,Z 10.501,A 0.015,B 0.000,C -180.000} C_DIS
LIN {X -399.721,Y 339.072,Z 10.500,A 0.015,B -0.000,C -180.000} C_DIS
LIN {X -400.552,Y 338.848,Z 10.470,A 0.015,B 0.000,C -180.000} C_DIS
LIN {X -400.596,Y 338.832,Z 10.468,A 0.015,B 0.000,C -180.000} C_DIS
LIN {X -401.281,Y 338.494,Z 10.442,A 0.015,B 0.000,C -180.000} C_DIS
LIN {X -401.404,Y 338.418,Z 10.436,A 0.015,B -0.000,C 180.000} C_DIS
LIN {X -402.842,Y 337.053,Z 10.367,A 0.015,B 0.000,C 180.000} C_DIS
LIN {X -402.866,Y 337.018,Z 10.365,A 0.015,B 0.000,C -180.000} C_DIS
LIN {X -403.753,Y 334.430,Z 10.269,A 0.015,B -0.000,C -180.000} C_DIS
LIN {X -403.779,Y 333.946,Z 10.252,A 0.015,B -0.000,C 180.000} C_DIS
LIN {X -403.787,Y 333.653,Z 10.241,A 0.015,B -0.000,C 180.000} C_DIS
LIN {X -403.787,Y 333.050,Z 10.220,A 0.015,B 0.000,C -180.000} C_DIS
LIN {X -401.252,Y 328.076,Z 10.018,A 0.015,B -0.000,C 180.000} C_DIS
LIN {X -395.738,Y 327.203,Z 9.816,A 0.015,B -0.000,C -180.000} C_DIS
LIN {X -391.790,Y 331.150,Z 9.613,A 0.015,B 0.000,C -180.000} C_DIS
LIN {X -392.664,Y 336.664,Z 9.411,A 0.015,B -0.000,C -180.000} C_DIS
LIN {X -397.638,Y 339.199,Z 9.208,A 0.015,B -0.000,C -180.000} C_DIS
LIN {X -398.507,Y 339.199,Z 9.178,A 0.015,B 0.000,C -180.000} C_DIS
LIN {X -399.336,Y 339.133,Z 9.149,A 0.015,B 0.000,C -180.000} C_DIS
LIN {X -399.692,Y 339.076,Z 9.136,A 0.015,B 0.000,C -180.000} C_DIS
LIN {X -400.552,Y 338.848,Z 9.105,A 0.015,B 0.000,C -180.000} C_DIS
LIN {X -400.596,Y 338.832,Z 9.104,A 0.015,B -0.000,C -180.000} C_DIS
LIN {X -401.281,Y 338.494,Z 9.077,A 0.015,B -0.000,C 180.000} C_DIS
LIN {X -401.404,Y 338.418,Z 9.072,A 0.015,B 0.000,C 180.000} C_DIS
LIN {X -402.842,Y 337.053,Z 9.002,A 0.015,B 0.000,C 180.000} C_DIS
LIN {X -402.866,Y 337.018,Z 9.001,A 0.015,B -0.000,C -180.000} C_DIS
LIN {X -403.753,Y 334.430,Z 8.904,A 0.015,B 0.000,C 180.000} C_DIS
LIN {X -403.779,Y 333.946,Z 8.887,A 0.015,B -0.000,C -180.000} C_DIS
LIN {X -403.787,Y 333.653,Z 8.877,A 0.015,B 0.000,C -180.000} C_DIS
LIN {X -403.787,Y 333.050,Z 8.856,A 0.015,B -0.000,C -180.000} C_DIS
LIN {X -401.252,Y 328.076,Z 8.653,A 0.015,B -0.000,C -180.000} C_DIS
LIN {X -395.738,Y 327.203,Z 8.451,A 0.015,B 0.000,C 180.000} C_DIS
LIN {X -391.790,Y 331.150,Z 8.249,A 0.015,B 0.000,C -180.000} C_DIS
LIN {X -392.664,Y 336.664,Z 8.046,A 0.015,B 0.000,C -180.000} C_DIS
LIN {X -397.638,Y 339.199,Z 7.844,A 0.015,B -0.000,C -180.000} C_DIS
LIN {X -398.507,Y 339.199,Z 7.814,A 0.015,B -0.000,C -180.000} C_DIS
LIN {X -399.336,Y 339.133,Z 7.785,A 0.015,B -0.000,C 180.000} C_DIS
LIN {X -399.692,Y 339.076,Z 7.772,A 0.015,B -0.000,C -180.000} C_DIS
LIN {X -400.552,Y 338.848,Z 7.741,A 0.015,B 0.000,C -180.000} C_DIS
LIN {X -400.596,Y 338.832,Z 7.739,A 0.015,B -0.000,C -180.000} C_DIS
LIN {X -401.281,Y 338.494,Z 7.712,A 0.015,B -0.000,C -180.000} C_DIS
LIN {X -401.404,Y 338.418,Z 7.707,A 0.015,B -0.000,C 180.000} C_DIS
LIN {X -402.842,Y 337.053,Z 7.638,A 0.015,B 0.000,C -180.000} C_DIS
LIN {X -402.866,Y 337.018,Z 7.636,A 0.015,B 0.000,C -180.000} C_DIS
LIN {X -403.753,Y 334.430,Z 7.539,A 0.015,B 0.000,C -180.000} C_DIS
LIN {X -403.779,Y 333.946,Z 7.522,A 0.015,B 0.000,C 180.000} C_DIS
LIN {X -403.787,Y 333.653,Z 7.512,A 0.015,B -0.000,C -180.000} C_DIS
LIN {X -403.787,Y 333.050,Z 7.491,A 0.015,B 0.000,C -180.000} C_DIS
LIN {X -401.252,Y 328.076,Z 7.289,A 0.015,B -0.000,C -180.000} C_DIS
LIN {X -395.738,Y 327.203,Z 7.086,A 0.015,B 0.000,C -180.000} C_DIS
LIN {X -391.790,Y 331.150,Z 6.884,A 0.015,B -0.000,C -180.000} C_DIS
LIN {X -392.664,Y 336.664,Z 6.682,A 0.015,B 0.000,C -180.000} C_DIS
LIN {X -397.638,Y 339.199,Z 6.479,A 0.015,B 0.000,C 180.000} C_DIS
LIN {X -398.507,Y 339.199,Z 6.449,A 0.015,B 0.000,C -180.000} C_DIS
LIN {X -399.336,Y 339.133,Z 6.420,A 0.015,B -0.000,C 180.000} C_DIS
LIN {X -399.692,Y 339.076,Z 6.407,A 0.015,B -0.000,C -180.000} C_DIS
LIN {X -400.552,Y 338.848,Z 6.376,A 0.015,B -0.000,C -180.000} C_DIS
LIN {X -400.596,Y 338.832,Z 6.375,A 0.015,B 0.000,C -180.000} C_DIS
LIN {X -401.281,Y 338.494,Z 6.348,A 0.015,B 0.000,C -180.000} C_DIS
LIN {X -401.404,Y 338.418,Z 6.343,A 0.015,B 0.000,C -180.000} C_DIS
LIN {X -402.842,Y 337.053,Z 6.273,A 0.015,B -0.000,C 180.000} C_DIS
LIN {X -402.866,Y 337.018,Z 6.272,A 0.015,B -0.000,C -180.000} C_DIS
LIN {X -403.753,Y 334.430,Z 6.175,A 0.015,B 0.000,C -180.000} C_DIS
LIN {X -403.779,Y 333.946,Z 6.158,A 0.015,B 0.000,C -180.000} C_DIS
LIN {X -403.787,Y 333.653,Z 6.148,A 0.015,B 0.000,C -180.000} C_DIS
LIN {X -403.787,Y 333.050,Z 6.127,A 0.015,B -0.000,C -180.000} C_DIS
LIN {X -401.252,Y 328.076,Z 5.924,A 0.015,B 0.000,C -180.000} C_DIS
LIN {X -395.738,Y 327.203,Z 5.722,A 0.015,B -0.000,C -180.000} C_DIS
LIN {X -391.790,Y 331.150,Z 5.520,A 0.015,B -0.000,C -180.000} C_DIS
LIN {X -392.664,Y 336.664,Z 5.317,A 0.015,B -0.000,C 180.000} C_DIS
LIN {X -397.638,Y 339.199,Z 5.115,A 0.015,B 0.000,C -180.000} C_DIS
LIN {X -398.507,Y 339.199,Z 5.084,A 0.015,B 0.000,C -180.000} C_DIS
LIN {X -399.336,Y 339.133,Z 5.055,A 0.015,B 0.000,C -180.000} C_DIS
LIN {X -399.692,Y 339.076,Z 5.043,A 0.015,B 0.000,C -180.000} C_DIS
LIN {X -400.552,Y 338.848,Z 5.012,A 0.015,B 0.000,C 180.000} C_DIS
LIN {X -400.596,Y 338.832,Z 5.010,A 0.015,B 0.000,C -180.000} C_DIS
LIN {X -401.281,Y 338.494,Z 4.983,A 0.015,B -0.000,C -180.000} C_DIS
LIN {X -401.404,Y 338.418,Z 4.978,A 0.015,B -0.000,C -180.000} C_DIS
LIN {X -402.842,Y 337.053,Z 4.909,A 0.015,B -0.000,C -180.000} C_DIS
LIN {X -402.866,Y 337.018,Z 4.907,A 0.015,B 0.000,C 180.000} C_DIS
LIN {X -403.753,Y 334.430,Z 4.810,A 0.015,B -0.000,C -180.000} C_DIS
LIN {X -403.779,Y 333.946,Z 4.793,A 0.015,B 0.000,C -180.000} C_DIS
LIN {X -403.787,Y 333.653,Z 4.783,A 0.015,B -0.000,C 180.000} C_DIS
LIN {X -403.787,Y 333.050,Z 4.762,A 0.015,B -0.000,C 180.000} C_DIS
LIN {X -401.252,Y 328.076,Z 4.560,A 0.015,B 0.000,C 180.000} C_DIS
LIN {X -395.738,Y 327.203,Z 4.357,A 0.015,B -0.000,C -180.000} C_DIS
LIN {X -391.790,Y 331.150,Z 4.155,A 0.015,B -0.000,C 180.000} C_DIS
LIN {X -392.664,Y 336.664,Z 3.953,A 0.015,B -0.000,C 180.000} C_DIS
LIN {X -397.638,Y 339.199,Z 3.750,A 0.015,B -0.000,C 180.000} C_DIS
LIN {X -398.507,Y 339.199,Z 3.720,A 0.015,B 0.000,C 180.000} C_DIS
LIN {X -399.336,Y 339.133,Z 3.691,A 0.015,B -0.000,C -180.000} C_DIS
LIN {X -399.692,Y 339.076,Z 3.678,A 0.015,B -0.000,C -180.000} C_DIS
LIN {X -400.552,Y 338.848,Z 3.647,A 0.015,B -0.000,C -180.000} C_DIS
LIN {X -400.596,Y 338.832,Z 3.646,A 0.015,B -0.000,C -180.000} C_DIS
LIN {X -401.281,Y 338.494,Z 3.619,A 0.015,B -0.000,C -180.000} C_DIS
LIN {X -401.404,Y 338.418,Z 3.614,A 0.015,B -0.000,C 180.000} C_DIS
LIN {X -402.842,Y 337.053,Z 3.544,A 0.015,B 0.000,C -180.000} C_DIS
LIN {X -402.866,Y 337.018,Z 3.543,A 0.015,B 0.000,C -180.000} C_DIS
LIN {X -403.753,Y 334.430,Z 3.446,A 0.015,B 0.000,C -180.000} C_DIS
LIN {X -403.779,Y 333.946,Z 3.429,A 0.015,B 0.000,C -180.000} C_DIS
LIN {X -403.787,Y 333.653,Z 3.419,A 0.015,B -0.000,C -180.000} C_DIS
LIN {X -403.787,Y 333.050,Z 3.398,A 0.015,B 0.000,C -180.000} C_DIS
LIN {X -401.252,Y 328.076,Z 3.195,A 0.015,B -0.000,C -180.000} C_DIS
LIN {X -395.738,Y 327.203,Z 2.993,A 0.015,B -0.000,C -180.000} C_DIS
LIN {X -391.790,Y 331.150,Z 2.790,A 0.015,B -0.000,C -180.000} C_DIS
LIN {X -392.664,Y 336.664,Z 2.588,A 0.015,B -0.000,C 180.000} C_DIS
LIN {X -397.638,Y 339.199,Z 2.386,A 0.015,B 0.000,C -180.000} C_DIS
LIN {X -398.507,Y 339.199,Z 2.355,A 0.015,B 0.000,C -180.000} C_DIS
LIN {X -399.336,Y 339.133,Z 2.326,A 0.015,B 0.000,C 180.000} C_DIS
LIN {X -399.692,Y 339.076,Z 2.314,A 0.015,B -0.000,C -180.000} C_DIS
LIN {X -400.552,Y 338.848,Z 2.283,A 0.015,B -0.000,C -180.000} C_DIS
LIN {X -400.596,Y 338.832,Z 2.281,A 0.015,B 0.000,C 180.000} C_DIS
LIN {X -401.281,Y 338.494,Z 2.254,A 0.015,B 0.000,C 180.000} C_DIS
LIN {X -401.404,Y 338.418,Z 2.249,A 0.015,B -0.000,C -180.000} C_DIS
LIN {X -402.842,Y 337.053,Z 2.179,A 0.015,B 0.000,C -180.000} C_DIS
LIN {X -402.866,Y 337.018,Z 2.178,A 0.015,B -0.000,C -180.000} C_DIS
LIN {X -403.753,Y 334.430,Z 2.081,A 0.015,B -0.000,C 180.000} C_DIS
LIN {X -403.779,Y 333.946,Z 2.064,A 0.015,B 0.000,C -180.000} C_DIS
LIN {X -403.787,Y 333.653,Z 2.054,A 0.015,B 0.000,C 180.000} C_DIS
LIN {X -403.787,Y 333.050,Z 2.033,A 0.015,B -0.000,C 180.000} C_DIS
LIN {X -401.252,Y 328.076,Z 1.831,A 0.015,B 0.000,C -180.000} C_DIS
LIN {X -395.738,Y 327.203,Z 1.628,A 0.015,B -0.000,C 180.000} C_DIS
LIN {X -391.790,Y 331.150,Z 1.426,A 0.015,B 0.000,C -180.000} C_DIS
LIN {X -392.664,Y 336.664,Z 1.224,A 0.015,B -0.000,C -180.000} C_DIS
LIN {X -397.638,Y 339.199,Z 1.021,A 0.015,B -0.000,C -180.000} C_DIS
LIN {X -398.507,Y 339.199,Z 0.991,A 0.015,B 0.000,C -180.000} C_DIS
LIN {X -399.336,Y 339.133,Z 0.962,A 0.015,B -0.000,C 180.000} C_DIS
LIN {X -399.692,Y 339.076,Z 0.949,A 0.015,B -0.000,C -180.000} C_DIS
LIN {X -400.552,Y 338.848,Z 0.918,A 0.015,B -0.000,C -180.000} C_DIS
LIN {X -400.596,Y 338.832,Z 0.916,A 0.015,B 0.000,C -180.000} C_DIS
LIN {X -401.281,Y 338.494,Z 0.890,A 0.015,B 0.000,C 180.000} C_DIS
LIN {X -401.404,Y 338.418,Z 0.885,A 0.015,B -0.000,C -180.000} C_DIS
LIN {X -402.842,Y 337.053,Z 0.815,A 0.015,B 0.000,C 180.000} C_DIS
LIN {X -402.866,Y 337.018,Z 0.813,A 0.015,B -0.000,C -180.000} C_DIS
LIN {X -403.753,Y 334.430,Z 0.717,A 0.015,B -0.000,C -180.000} C_DIS
LIN {X -403.779,Y 333.946,Z 0.700,A 0.015,B 0.000,C 180.000} C_DIS
LIN {X -403.787,Y 333.653,Z 0.690,A 0.015,B 0.000,C 180.000} C_DIS
LIN {X -403.787,Y 333.050,Z 0.668,A 0.015,B -0.000,C -180.000} C_DIS
LIN {X -401.252,Y 328.076,Z 0.466,A 0.015,B 0.000,C -180.000} C_DIS
LIN {X -395.738,Y 327.203,Z 0.264,A 0.015,B -0.000,C -180.000} C_DIS
LIN {X -391.790,Y 331.150,Z 0.061,A 0.015,B 0.000,C 180.000} C_DIS
LIN {X -392.664,Y 336.664,Z -0.141,A 0.015,B -0.000,C -180.000} C_DIS
LIN {X -397.638,Y 339.199,Z -0.343,A 0.015,B 0.000,C -180.000} C_DIS
LIN {X -398.507,Y 339.199,Z -0.374,A 0.015,B 0.000,C -180.000} C_DIS
LIN {X -399.336,Y 339.133,Z -0.403,A 0.015,B 0.000,C -180.000} C_DIS
LIN {X -399.692,Y 339.076,Z -0.415,A 0.015,B 0.000,C 180.000} C_DIS
LIN {X -400.552,Y 338.848,Z -0.447,A 0.015,B -0.000,C -180.000} C_DIS
LIN {X -400.596,Y 338.832,Z -0.448,A 0.015,B 0.000,C -180.000} C_DIS
LIN {X -401.281,Y 338.494,Z -0.475,A 0.015,B 0.000,C -180.000} C_DIS
LIN {X -401.404,Y 338.418,Z -0.480,A 0.015,B 0.000,C -180.000} C_DIS
LIN {X -402.842,Y 337.053,Z -0.550,A 0.015,B 0.000,C -180.000} C_DIS
LIN {X -402.866,Y 337.018,Z -0.551,A 0.015,B -0.000,C -180.000} C_DIS
LIN {X -403.753,Y 334.430,Z -0.648,A 0.015,B -0.000,C 180.000} C_DIS
LIN {X -403.779,Y 333.946,Z -0.665,A 0.015,B -0.000,C 180.000} C_DIS
LIN {X -403.787,Y 333.653,Z -0.675,A 0.015,B -0.000,C -180.000} C_DIS
LIN {X -403.787,Y 333.050,Z -0.696,A 0.015,B -0.000,C -180.000} C_DIS
LIN {X -401.252,Y 328.076,Z -0.898,A 0.015,B 0.000,C -180.000} C_DIS
LIN {X -395.738,Y 327.203,Z -1.101,A 0.015,B -0.000,C 180.000} C_DIS
LIN {X -391.790,Y 331.150,Z -1.303,A 0.015,B 0.000,C -180.000} C_DIS
LIN {X -392.664,Y 336.664,Z -1.506,A 0.015,B 0.000,C -180.000} C_DIS
LIN {X -397.638,Y 339.199,Z -1.708,A 0.015,B 0.000,C 180.000} C_DIS
LIN {X -398.507,Y 339.199,Z -1.738,A 0.015,B -0.000,C -180.000} C_DIS
LIN {X -399.336,Y 339.133,Z -1.767,A 0.015,B -0.000,C -180.000} C_DIS
LIN {X -399.692,Y 339.076,Z -1.780,A 0.015,B -0.000,C -180.000} C_DIS
LIN {X -400.552,Y 338.848,Z -1.811,A 0.015,B -0.000,C -180.000} C_DIS
LIN {X -400.596,Y 338.832,Z -1.813,A 0.015,B -0.000,C -180.000} C_DIS
LIN {X -401.281,Y 338.494,Z -1.839,A 0.015,B 0.000,C 180.000} C_DIS
LIN {X -401.404,Y 338.418,Z -1.844,A 0.015,B -0.000,C -180.000} C_DIS
LIN {X -402.842,Y 337.053,Z -1.914,A 0.015,B 0.000,C -180.000} C_DIS
LIN {X -402.866,Y 337.018,Z -1.916,A 0.015,B 0.000,C 180.000} C_DIS
LIN {X -403.753,Y 334.430,Z -2.012,A 0.015,B 0.000,C 180.000} C_DIS
LIN {X -403.779,Y 333.946,Z -2.029,A 0.015,B -0.000,C -180.000} C_DIS
LIN {X -403.787,Y 333.653,Z -2.040,A 0.015,B 0.000,C -180.000} C_DIS
LIN {X -403.787,Y 333.050,Z -2.061,A 0.015,B 0.000,C -180.000} C_DIS
LIN {X -401.252,Y 328.076,Z -2.263,A 0.015,B -0.000,C -180.000} C_DIS
LIN {X -395.738,Y 327.203,Z -2.465,A 0.015,B -0.000,C -180.000} C_DIS
LIN {X -391.790,Y 331.150,Z -2.668,A 0.015,B 0.000,C 180.000} C_DIS
LIN {X -392.664,Y 336.664,Z -2.870,A 0.015,B 0.000,C 180.000} C_DIS
LIN {X -397.638,Y 339.199,Z -3.072,A 0.015,B 0.000,C -180.000} C_DIS
LIN {X -398.507,Y 339.199,Z -3.103,A 0.015,B -0.000,C -180.000} C_DIS
LIN {X -399.336,Y 339.133,Z -3.132,A 0.015,B 0.000,C -180.000} C_DIS
LIN {X -399.692,Y 339.076,Z -3.145,A 0.015,B 0.000,C 180.000} C_DIS
LIN {X -400.552,Y 338.848,Z -3.176,A 0.015,B -0.000,C -180.000} C_DIS
LIN {X -400.596,Y 338.832,Z -3.177,A 0.015,B 0.000,C -180.000} C_DIS
LIN {X -401.281,Y 338.494,Z -3.204,A 0.015,B 0.000,C -180.000} C_DIS
LIN {X -401.404,Y 338.418,Z -3.209,A 0.015,B 0.000,C -180.000} C_DIS
LIN {X -402.842,Y 337.053,Z -3.279,A 0.015,B -0.000,C -180.000} C_DIS
LIN {X -402.866,Y 337.018,Z -3.280,A 0.015,B -0.000,C -180.000} C_DIS
LIN {X -403.753,Y 334.430,Z -3.377,A 0.015,B -0.000,C -180.000} C_DIS
LIN {X -403.779,Y 333.946,Z -3.394,A 0.015,B -0.000,C -180.000} C_DIS
LIN {X -403.787,Y 333.653,Z -3.404,A 0.015,B -0.000,C 180.000} C_DIS
LIN {X -403.787,Y 333.050,Z -3.425,A 0.015,B -0.000,C 180.000} C_DIS
LIN {X -401.252,Y 328.076,Z -3.628,A 0.015,B 0.000,C -180.000} C_DIS
LIN {X -395.738,Y 327.203,Z -3.830,A 0.015,B -0.000,C -180.000} C_DIS
LIN {X -391.790,Y 331.150,Z -4.032,A 0.015,B -0.000,C -180.000} C_DIS
LIN {X -392.664,Y 336.664,Z -4.235,A 0.015,B -0.000,C 180.000} C_DIS
LIN {X -397.638,Y 339.199,Z -4.437,A 0.015,B 0.000,C 180.000} C_DIS
LIN {X -398.507,Y 339.199,Z -4.467,A 0.015,B 0.000,C 180.000} C_DIS
LIN {X -399.336,Y 339.133,Z -4.496,A 0.015,B 0.000,C -180.000} C_DIS
LIN {X -399.692,Y 339.076,Z -4.509,A 0.015,B -0.000,C 180.000} C_DIS
LIN {X -400.552,Y 338.848,Z -4.540,A 0.015,B 0.000,C -180.000} C_DIS
LIN {X -400.596,Y 338.832,Z -4.542,A 0.015,B 0.000,C -180.000} C_DIS
LIN {X -401.281,Y 338.494,Z -4.569,A 0.015,B -0.000,C -180.000} C_DIS
LIN {X -401.404,Y 338.418,Z -4.574,A 0.015,B 0.000,C -180.000} C_DIS
LIN {X -402.842,Y 337.053,Z -4.643,A 0.015,B -0.000,C 180.000} C_DIS
LIN {X -402.866,Y 337.018,Z -4.645,A 0.015,B -0.000,C -180.000} C_DIS
LIN {X -403.753,Y 334.430,Z -4.742,A 0.015,B 0.000,C -180.000} C_DIS
LIN {X -403.779,Y 333.946,Z -4.758,A 0.015,B 0.000,C -180.000} C_DIS
LIN {X -403.787,Y 333.653,Z -4.769,A 0.015,B -0.000,C -180.000} C_DIS
LIN {X -403.787,Y 333.050,Z -4.790,A 0.015,B 0.000,C -180.000} C_DIS
LIN {X -401.252,Y 328.076,Z -4.992,A 0.015,B 0.000,C 180.000} C_DIS
LIN {X -395.738,Y 327.203,Z -5.195,A 0.015,B 0.000,C -180.000} C_DIS
LIN {X -391.790,Y 331.150,Z -5.397,A 0.015,B -0.000,C -180.000} C_DIS
LIN {X -392.664,Y 336.664,Z -5.599,A 0.015,B -0.000,C -180.000} C_DIS
LIN {X -397.638,Y 339.199,Z -5.802,A 0.015,B -0.000,C 180.000} C_DIS
LIN {X -398.507,Y 339.199,Z -5.832,A 0.015,B 0.000,C 180.000} C_DIS
LIN {X -399.336,Y 339.133,Z -5.861,A 0.015,B 0.000,C -180.000} C_DIS
LIN {X -399.692,Y 339.076,Z -5.874,A 0.015,B 0.000,C -180.000} C_DIS
LIN {X -400.552,Y 338.848,Z -5.905,A 0.015,B -0.000,C -180.000} C_DIS
LIN {X -400.596,Y 338.832,Z -5.906,A 0.015,B 0.000,C -180.000} C_DIS
LIN {X -401.281,Y 338.494,Z -5.933,A 0.015,B -0.000,C 180.000} C_DIS
LIN {X -401.404,Y 338.418,Z -5.938,A 0.015,B 0.000,C 180.000} C_DIS
LIN {X -402.842,Y 337.053,Z -6.008,A 0.015,B 0.000,C -180.000} C_DIS
LIN {X -402.866,Y 337.018,Z -6.009,A 0.015,B 0.000,C -180.000} C_DIS
LIN {X -403.753,Y 334.430,Z -6.106,A 0.015,B -0.000,C -180.000} C_DIS
LIN {X -403.779,Y 333.946,Z -6.123,A 0.015,B 0.000,C -180.000} C_DIS
LIN {X -403.787,Y 333.653,Z -6.133,A 0.015,B 0.000,C -180.000} C_DIS
LIN {X -403.787,Y 333.050,Z -6.154,A 0.015,B -0.000,C 180.000} C_DIS
LIN {X -401.252,Y 328.076,Z -6.357,A 0.015,B 0.000,C 180.000} C_DIS
LIN {X -395.738,Y 327.203,Z -6.559,A 0.015,B -0.000,C 180.000} C_DIS
LIN {X -391.790,Y 331.150,Z -6.761,A 0.015,B 0.000,C -180.000} C_DIS
LIN {X -392.664,Y 336.664,Z -6.964,A 0.015,B 0.000,C -180.000} C_DIS
LIN {X -397.638,Y 339.199,Z -7.166,A 0.015,B -0.000,C -180.000} C_DIS
LIN {X -398.507,Y 339.199,Z -7.196,A 0.015,B -0.000,C -180.000} C_DIS
LIN {X -399.336,Y 339.133,Z -7.226,A 0.015,B 0.000,C -180.000} C_DIS
LIN {X -399.692,Y 339.076,Z -7.238,A 0.015,B 0.000,C 180.000} C_DIS
LIN {X -400.552,Y 338.848,Z -7.269,A 0.015,B 0.000,C -180.000} C_DIS
LIN {X -400.596,Y 338.832,Z -7.271,A 0.015,B 0.000,C -180.000} C_DIS
LIN {X -401.281,Y 338.494,Z -7.298,A 0.015,B -0.000,C 180.000} C_DIS
LIN {X -401.404,Y 338.418,Z -7.303,A 0.015,B 0.000,C 180.000} C_DIS
LIN {X -402.842,Y 337.053,Z -7.372,A 0.015,B 0.000,C -180.000} C_DIS
LIN {X -402.866,Y 337.018,Z -7.374,A 0.015,B 0.000,C -180.000} C_DIS
LIN {X -403.753,Y 334.430,Z -7.471,A 0.015,B -0.000,C 180.000} C_DIS
LIN {X -403.779,Y 333.946,Z -7.488,A 0.015,B -0.000,C -180.000} C_DIS
LIN {X -403.787,Y 333.653,Z -7.498,A 0.015,B 0.000,C -180.000} C_DIS
LIN {X -403.787,Y 333.050,Z -7.519,A 0.015,B 0.000,C -180.000} C_DIS
LIN {X -401.252,Y 328.076,Z -7.721,A 0.015,B -0.000,C -180.000} C_DIS
LIN {X -395.738,Y 327.203,Z -7.924,A 0.015,B 0.000,C 180.000} C_DIS
LIN {X -391.790,Y 331.150,Z -8.126,A 0.015,B 0.000,C -180.000} C_DIS
LIN {X -392.664,Y 336.664,Z -8.328,A 0.015,B -0.000,C 180.000} C_DIS
LIN {X -397.638,Y 339.199,Z -8.531,A 0.015,B 0.000,C -180.000} C_DIS
LIN {X -398.507,Y 339.199,Z -8.561,A 0.015,B 0.000,C 180.000} C_DIS
LIN {X -399.336,Y 339.133,Z -8.590,A 0.015,B 0.000,C 180.000} C_DIS
LIN {X -399.692,Y 339.076,Z -8.603,A 0.015,B 0.000,C -180.000} C_DIS
LIN {X -400.552,Y 338.848,Z -8.634,A 0.015,B -0.000,C -180.000} C_DIS
LIN {X -400.596,Y 338.832,Z -8.635,A 0.015,B -0.000,C -180.000} C_DIS
LIN {X -401.281,Y 338.494,Z -8.662,A 0.015,B -0.000,C -180.000} C_DIS
LIN {X -401.404,Y 338.418,Z -8.667,A 0.015,B -0.000,C -180.000} C_DIS
LIN {X -402.842,Y 337.053,Z -8.737,A 0.015,B -0.000,C -180.000} C_DIS
LIN {X -402.866,Y 337.018,Z -8.738,A 0.015,B -0.000,C -180.000} C_DIS
LIN {X -403.753,Y 334.430,Z -8.835,A 0.015,B 0.000,C 180.000} C_DIS
LIN {X -403.779,Y 333.946,Z -8.852,A 0.015,B -0.000,C -180.000} C_DIS
LIN {X -403.787,Y 333.653,Z -8.862,A 0.015,B 0.000,C -180.000} C_DIS
LIN {X -403.787,Y 333.050,Z -8.883,A 0.015,B 0.000,C -180.000} C_DIS
LIN {X -401.252,Y 328.076,Z -9.086,A 0.015,B 0.000,C 180.000} C_DIS
LIN {X -395.738,Y 327.203,Z -9.288,A 0.015,B 0.000,C 180.000} C_DIS
LIN {X -391.790,Y 331.150,Z -9.491,A 0.015,B 0.000,C -180.000} C_DIS
LIN {X -392.664,Y 336.664,Z -9.693,A 0.015,B -0.000,C 180.000} C_DIS
LIN {X -397.638,Y 339.199,Z -9.895,A 0.015,B 0.000,C -180.000} C_DIS
LIN {X -398.507,Y 339.199,Z -9.926,A 0.015,B -0.000,C -180.000} C_DIS
LIN {X -399.336,Y 339.133,Z -9.955,A 0.015,B 0.000,C -180.000} C_DIS
LIN {X -399.692,Y 339.076,Z -9.967,A 0.015,B 0.000,C -180.000} C_DIS
LIN {X -400.552,Y 338.848,Z -9.998,A 0.015,B 0.000,C 180.000} C_DIS
LIN {X -400.596,Y 338.832,Z -10.000,A 0.015,B -0.000,C -180.000} C_DIS
LIN {X -400.134,Y 339.006,Z -10.000,A 0.015,B -0.000,C -180.000} C_DIS
LIN {X -398.924,Y 339.199,Z -10.000,A 0.015,B 0.000,C 180.000} C_DIS
LIN {X -213.124,Y 339.203,Z -10.000,A 0.015,B 0.000,C 180.000} C_DIS
LIN {X -213.229,Y 339.187,Z -10.000,A 0.015,B 0.000,C -180.000} C_DIS
LIN {X -213.439,Y 339.148,Z -10.000,A 0.015,B -0.000,C -180.000} C_DIS
LIN {X -214.528,Y 338.911,Z -10.000,A 0.015,B 0.000,C 180.000} C_DIS
LIN {X -215.300,Y 338.641,Z -10.000,A 0.015,B -0.000,C 180.000} C_DIS
LIN {X -225.821,Y 333.466,Z -10.000,A 0.015,B 0.000,C -180.000} C_DIS
LIN {X -225.999,Y 333.371,Z -10.000,A 0.015,B 0.000,C 180.000} C_DIS
LIN {X -227.450,Y 332.547,Z -10.000,A 0.015,B 0.000,C 180.000} C_DIS
LIN {X -228.124,Y 332.044,Z -10.000,A 0.015,B -0.000,C -180.000} C_DIS
LIN {X -237.248,Y 323.268,Z -10.000,A 0.015,B 0.000,C 180.000} C_DIS
LIN {X -237.617,Y 322.849,Z -10.000,A 0.015,B 0.000,C 180.000} C_DIS
LIN {X -238.156,Y 322.124,Z -10.000,A 0.015,B 0.000,C 180.000} C_DIS
LIN {X -238.415,Y 321.719,Z -10.000,A 0.015,B 0.000,C -180.000} C_DIS
LIN {X -243.932,Y 311.562,Z -10.000,A 0.015,B 0.000,C 180.000} C_DIS
LIN {X -244.052,Y 311.318,Z -10.000,A 0.015,B 0.000,C 180.000} C_DIS
LIN {X -244.695,Y 309.867,Z -10.000,A 0.015,B -0.000,C 180.000} C_DIS
LIN {X -244.946,Y 309.009,Z -10.000,A 0.015,B -0.000,C 180.000} C_DIS
LIN {X -246.389,Y 299.577,Z -10.000,A 0.015,B -0.000,C 180.000} C_DIS
LIN {X -246.415,Y 299.356,Z -10.000,A 0.015,B -0.000,C 180.000} C_DIS
LIN {X -246.509,Y 298.268,Z -10.000,A 0.015,B 0.000,C 180.000} C_DIS
CIRC {X -246.514,Y 297.746,Z -10.000,A 0.015,B -0.000,C -180.000},{X -246.438,Y 297.230,Z -10.000,A 0.015,B -0.000,C -180.000} C_DIS
LIN {X -245.040,Y 291.057,Z -10.000,A 0.015,B 0.000,C 180.000} C_DIS
LIN {X -245.029,Y 291.008,Z -10.000,A 0.015,B 0.000,C -180.000} C_DIS
LIN {X -244.063,Y 287.024,Z -10.000,A 0.015,B 0.000,C 180.000} C_DIS
LIN {X -243.781,Y 286.268,Z -10.000,A 0.015,B -0.000,C -180.000} C_DIS
LIN {X -243.052,Y 284.855,Z -10.000,A 0.015,B 0.000,C -180.000} C_DIS
LIN {X -242.815,Y 284.464,Z -10.000,A 0.015,B -0.000,C 180.000} C_DIS
LIN {X -238.705,Y 278.610,Z -10.000,A 0.015,B 0.000,C -180.000} C_DIS
LIN {X -238.576,Y 278.437,Z -10.000,A 0.015,B -0.000,C 180.000} C_DIS
LIN {X -237.131,Y 276.636,Z -10.000,A 0.015,B 0.000,C -180.000} C_DIS
LIN {X -236.639,Y 276.137,Z -10.000,A 0.015,B -0.000,C -180.000} C_DIS
LIN {X -235.910,Y 275.539,Z -10.000,A 0.015,B 0.000,C -180.000} C_DIS
LIN {X -235.625,Y 275.329,Z -10.000,A 0.015,B -0.000,C 180.000} C_DIS
LIN {X -229.091,Y 271.024,Z -10.000,A 0.015,B -0.000,C -180.000} C_DIS
LIN {X -228.907,Y 270.912,Z -10.000,A 0.015,B 0.000,C -180.000} C_DIS
LIN {X -227.329,Y 270.011,Z -10.000,A 0.015,B -0.000,C -180.000} C_DIS
LIN {X -226.814,Y 269.771,Z -10.000,A 0.015,B 0.000,C -180.000} C_DIS
LIN {X -225.490,Y 269.287,Z -10.000,A 0.015,B 0.000,C 180.000} C_DIS
LIN {X -224.979,Y 269.145,Z -10.000,A 0.015,B 0.000,C 180.000} C_DIS
LIN {X -219.174,Y 268.006,Z -10.000,A 0.015,B 0.000,C 180.000} C_DIS
LIN {X -219.056,Y 267.985,Z -10.000,A 0.015,B 0.000,C 180.000} C_DIS
LIN {X -215.428,Y 267.406,Z -10.000,A 0.015,B 0.000,C 180.000} C_DIS
LIN {X -214.896,Y 267.364,Z -10.000,A 0.015,B 0.000,C 180.000} C_DIS
LIN {X -179.343,Y 267.359,Z -10.000,A 0.015,B 0.000,C -180.000} C_DIS
LIN {X -179.133,Y 267.365,Z -10.000,A 0.015,B -0.000,C 180.000} C_DIS
LIN {X -177.682,Y 267.455,Z -10.000,A 0.015,B 0.000,C 180.000} C_DIS
LIN {X -177.276,Y 267.505,Z -10.000,A 0.015,B -0.000,C 180.000} C_DIS
LIN {X -169.294,Y 268.982,Z -10.000,A 0.015,B 0.000,C -180.000} C_DIS
LIN {X -169.033,Y 269.041,Z -10.000,A 0.015,B 0.000,C -180.000} C_DIS
LIN {X -167.645,Y 269.413,Z -10.000,A 0.015,B 0.000,C -180.000} C_DIS
LIN {X -167.180,Y 269.575,Z -10.000,A 0.015,B -0.000,C 180.000} C_DIS
LIN {X -166.124,Y 270.032,Z -10.000,A 0.015,B -0.000,C -180.000} C_DIS
LIN {X -165.641,Y 270.289,Z -10.000,A 0.015,B 0.000,C 180.000} C_DIS
LIN {X -158.653,Y 274.766,Z -10.000,A 0.015,B 0.000,C 180.000} C_DIS
LIN {X -158.463,Y 274.897,Z -10.000,A 0.015,B -0.000,C -180.000} C_DIS
LIN {X -157.370,Y 275.707,Z -10.000,A 0.015,B 0.000,C 180.000} C_DIS
LIN {X -156.906,Y 276.122,Z -10.000,A 0.015,B 0.000,C 180.000} C_DIS
LIN {X -155.765,Y 277.350,Z -10.000,A 0.015,B 0.000,C 180.000} C_DIS
LIN {X -155.487,Y 277.691,Z -10.000,A 0.015,B -0.000,C 180.000} C_DIS
LIN {X -150.927,Y 284.096,Z -10.000,A 0.015,B 0.000,C -180.000} C_DIS
LIN {X -150.703,Y 284.457,Z -10.000,A 0.015,B 0.000,C 180.000} C_DIS
LIN {X -149.756,Y 286.220,Z -10.000,A 0.015,B 0.000,C -180.000} C_DIS
LIN {X -149.445,Y 287.039,Z -10.000,A 0.015,B 0.000,C -180.000} C_DIS
LIN {X -147.118,Y 296.833,Z -10.000,A 0.015,B 0.000,C 180.000} C_DIS
LIN {X -147.031,Y 297.447,Z -10.000,A 0.015,B 0.000,C 180.000} C_DIS
LIN {X -146.995,Y 298.172,Z -10.000,A 0.015,B -0.000,C -180.000} C_DIS
LIN {X -147.027,Y 298.837,Z -10.000,A 0.015,B 0.000,C -180.000} C_DIS
LIN {X -148.481,Y 308.631,Z -10.000,A 0.015,B 0.000,C 180.000} C_DIS
LIN {X -148.607,Y 309.171,Z -10.000,A 0.015,B -0.000,C -180.000} C_DIS
LIN {X -148.957,Y 310.259,Z -10.000,A 0.015,B 0.000,C 180.000} C_DIS
LIN {X -149.203,Y 310.833,Z -10.000,A 0.015,B 0.000,C 180.000} C_DIS
LIN {X -155.095,Y 321.715,Z -10.000,A 0.015,B 0.000,C 180.000} C_DIS
LIN {X -155.356,Y 322.124,Z -10.000,A 0.015,B 0.000,C -180.000} C_DIS
LIN {X -155.895,Y 322.849,Z -10.000,A 0.015,B -0.000,C -180.000} C_DIS
LIN {X -156.254,Y 323.258,Z -10.000,A 0.015,B -0.000,C -180.000} C_DIS
LIN {X -163.730,Y 330.513,Z -10.000,A 0.015,B 0.000,C 180.000} C_DIS
LIN {X -163.846,Y 330.620,Z -10.000,A 0.015,B -0.000,C 180.000} C_DIS
